  gc_DbmTranslation_fr_Text1195 : WSTRING(13) := "Dmc Heartbeat";
  gc_DbmTranslation_fr_Text1196 : WSTRING(15) := "Power On Ok Dmc";
  gc_DbmTranslation_fr_Text1197 : WSTRING(16) := "Operationnal Dmc";
  gc_DbmTranslation_fr_Text1198 : WSTRING(18) := "Go To Operationnal";
  gc_DbmTranslation_fr_Text1199 : WSTRING(22) := "New Go To Operationnal";
  gc_DbmTranslation_fr_Text1200 : WSTRING(16) := "Send Command NMT";
  gc_DbmTranslation_fr_Text1201 : WSTRING(12) := "Step Raz Dmc";
  gc_DbmTranslation_fr_Text1202 : WSTRING(24) := "Command Raz Dmc On Going";
  gc_DbmTranslation_fr_Text1203 : WSTRING(22) := "Dig4 Input Command STO";
  gc_DbmTranslation_fr_Text1204 : WSTRING(20) := "Active Fault Raz Dmc";
  gc_DbmTranslation_fr_Text1205 : WSTRING(16) := "Active Fault Dmc";
  gc_DbmTranslation_fr_Text1206 : WSTRING(30) := "Delta Arm Angular Sensor state";
  gc_DbmTranslation_fr_Text1207 : WSTRING(30) := "Delta Arm Angular Sensor value";
  gc_DbmTranslation_fr_Text1208 : WSTRING(56) := "Delta Arm Angular Sensor with calibration scaling  value";
  gc_DbmTranslation_fr_Text1209 : WSTRING(41) := "Delta Arm Angular Sensor raw value Master";
  gc_DbmTranslation_fr_Text1210 : WSTRING(40) := "Delta Arm Angular Sensor raw value slave";
  gc_DbmTranslation_fr_Text1211 : WSTRING(30) := "Arrow Arm Angular Sensor state";
  gc_DbmTranslation_fr_Text1212 : WSTRING(30) := "Arrow Arm Angular Sensor value";
  gc_DbmTranslation_fr_Text1213 : WSTRING(56) := "Arrow Arm Angular Sensor with calibration scaling  value";
  gc_DbmTranslation_fr_Text1214 : WSTRING(34) := "Arrow Arm Angular Sensor raw value";
  gc_DbmTranslation_fr_Text1215 : WSTRING(30) := "Arrow Arm Angular Sensor state";
  gc_DbmTranslation_fr_Text1216 : WSTRING(15) := "Gas Gauge value";
  gc_DbmTranslation_fr_Text1217 : WSTRING(19) := "Gas Gauge raw value";
  gc_DbmTranslation_fr_Text1218 : WSTRING(11) := "Aru 1 state";
  gc_DbmTranslation_fr_Text1219 : WSTRING(15) := "Aru 1 raw value";
  gc_DbmTranslation_fr_Text1220 : WSTRING(11) := "Aru 2 state";
  gc_DbmTranslation_fr_Text1221 : WSTRING(15) := "Aru 2 raw value";
  gc_DbmTranslation_fr_Text1222 : WSTRING(32) := "Entry Telescope Fdc Sensor state";
  gc_DbmTranslation_fr_Text1223 : WSTRING(36) := "Entry Telescope Fdc Sensor raw value";
  gc_DbmTranslation_fr_Text1224 : WSTRING(36) := "Folded Delta Arm Sensor state switch";
  gc_DbmTranslation_fr_Text1225 : WSTRING(33) := "Folded Delta Arm Sensor raw value";
  gc_DbmTranslation_fr_Text1226 : WSTRING(35) := "Folded Boom Arm Sensor state switch";
  gc_DbmTranslation_fr_Text1227 : WSTRING(32) := "Folded Boom Arm Sensor raw value";
  gc_DbmTranslation_fr_Text1228 : WSTRING(33) := "Forcing Motor Regime state switch";
  gc_DbmTranslation_fr_Text1229 : WSTRING(30) := "Forcing Motor Regime raw value";
  gc_DbmTranslation_fr_Text1230 : WSTRING(24) := "Active Help state switch";
  gc_DbmTranslation_fr_Text1231 : WSTRING(21) := "Active Help raw value";
  gc_DbmTranslation_fr_Text1232 : WSTRING(25) := "Oil Pressure state swtich";
  gc_DbmTranslation_fr_Text1233 : WSTRING(22) := "Oil Pressure raw value";
  gc_DbmTranslation_fr_Text1234 : WSTRING(30) := "Water Temperature state switch";
  gc_DbmTranslation_fr_Text1235 : WSTRING(27) := "Water Temperature raw value";
  gc_DbmTranslation_fr_Text1236 : WSTRING(21) := "Stop Motor Info State";
  gc_DbmTranslation_fr_Text1237 : WSTRING(25) := "Stop Motor Info Raw value";
  gc_DbmTranslation_fr_Text1238 : WSTRING(26) := "Turret Post Selector State";
  gc_DbmTranslation_fr_Text1239 : WSTRING(30) := "Turret Post Selector Raw Value";
  gc_DbmTranslation_fr_Text1240 : WSTRING(25) := "Radio Post Selector State";
  gc_DbmTranslation_fr_Text1241 : WSTRING(29) := "Radio Post Selector Raw Value";
  gc_DbmTranslation_fr_Text1242 : WSTRING(27) := "Nacelle Post Selector State";
  gc_DbmTranslation_fr_Text1243 : WSTRING(31) := "Nacelle Post Selector Raw Value";
  gc_DbmTranslation_fr_Text1244 : WSTRING(43) := "Regime motor alternator rotation per minute";
  gc_DbmTranslation_fr_Text1245 : WSTRING(26) := "Alternator charge ok state";
  gc_DbmTranslation_fr_Text1246 : WSTRING(26) := "Alternator charge ok value";
  gc_DbmTranslation_fr_Text1247 : WSTRING(35) := "Transmission1 Pressure Sensor State";
  gc_DbmTranslation_fr_Text1248 : WSTRING(35) := "Transmission1 Pressure Sensor Value";
  gc_DbmTranslation_fr_Text1249 : WSTRING(35) := "Transmission2 Pressure Sensor State";
  gc_DbmTranslation_fr_Text1250 : WSTRING(35) := "Transmission2 Pressure Sensor Value";
  gc_DbmTranslation_fr_Text1251 : WSTRING(25) := "Fault Pvg Delta Arm state";
  gc_DbmTranslation_fr_Text1252 : WSTRING(29) := "Fault Pvg Delta Arm raw value";
  gc_DbmTranslation_fr_Text1253 : WSTRING(24) := "Fault Pvg Boom Arm state";
  gc_DbmTranslation_fr_Text1254 : WSTRING(28) := "Fault Pvg Boom Arm raw value";
  gc_DbmTranslation_fr_Text1255 : WSTRING(29) := "Fault Pvg Telescope Arm state";
  gc_DbmTranslation_fr_Text1256 : WSTRING(33) := "Fault Pvg Telescope Arm raw value";
  gc_DbmTranslation_fr_Text1257 : WSTRING(26) := "Fault Pvg Ev Pro TOR state";
  gc_DbmTranslation_fr_Text1258 : WSTRING(30) := "Fault Pvg Ev Pro TOR raw value";
  gc_DbmTranslation_fr_Text1259 : WSTRING(28) := "Bypass Pressure Sensor State";
  gc_DbmTranslation_fr_Text1260 : WSTRING(28) := "Bypass Pressure Sensor Value";
  gc_DbmTranslation_fr_Text1261 : WSTRING(31) := "Bypass Pressure Sensor RawValue";
  gc_DbmTranslation_fr_Text1262 : WSTRING(19) := "Starter Motor State";
  gc_DbmTranslation_fr_Text1263 : WSTRING(23) := "Starter Motor Raw value";
  gc_DbmTranslation_fr_Text1264 : WSTRING(33) := "Oil Tank Temperature Sensor State";
  gc_DbmTranslation_fr_Text1265 : WSTRING(33) := "Oil Tank Temperature Sensor Value";
  gc_DbmTranslation_fr_Text1266 : WSTRING(37) := "Oil Tank Temperature Sensor Raw value";
  gc_DbmTranslation_fr_Text1267 : WSTRING(17) := "Blue Fire command";
  gc_DbmTranslation_fr_Text1268 : WSTRING(22) := "Blue Fire actual value";
  gc_DbmTranslation_fr_Text1269 : WSTRING(29) := "Orange Flashing Light command";
  gc_DbmTranslation_fr_Text1270 : WSTRING(34) := "Orange Flashing Light actual value";
  gc_DbmTranslation_fr_Text1271 : WSTRING(20) := "Anti Startup command";
  gc_DbmTranslation_fr_Text1272 : WSTRING(18) := "Anti Startup Value";
  gc_DbmTranslation_fr_Text1273 : WSTRING(18) := "Stop Motor command";
  gc_DbmTranslation_fr_Text1274 : WSTRING(15) := "Warming command";
  gc_DbmTranslation_fr_Text1275 : WSTRING(17) := "Ev Bypass command";
  gc_DbmTranslation_fr_Text1276 : WSTRING(21) := "EvBypass actual value";
  gc_DbmTranslation_fr_Text1277 : WSTRING(28) := "Supply Pvg Delta Arm command";
  gc_DbmTranslation_fr_Text1278 : WSTRING(33) := "Supply Pvg Delta Arm actual value";
  gc_DbmTranslation_fr_Text1279 : WSTRING(28) := "Supply Pvg Arrow Arm command";
  gc_DbmTranslation_fr_Text1280 : WSTRING(33) := "Supply Pvg Arrow Arm actual value";
  gc_DbmTranslation_fr_Text1281 : WSTRING(32) := "Supply Pvg Telescope Arm command";
  gc_DbmTranslation_fr_Text1282 : WSTRING(37) := "Supply Pvg Telescope Arm actual value";
  gc_DbmTranslation_fr_Text1283 : WSTRING(30) := "Supply Pvg Prop Ev TOR command";
  gc_DbmTranslation_fr_Text1284 : WSTRING(35) := "Supply Pvg Prop Ev TOR actual value";
  gc_DbmTranslation_fr_Text1285 : WSTRING(33) := "Ev Prop Motor Accelerator command";
  gc_DbmTranslation_fr_Text1286 : WSTRING(23) := "Ev Prop Generator state";
  gc_DbmTranslation_fr_Text1287 : WSTRING(25) := "Ev Prop Generator command";
  gc_DbmTranslation_fr_Text1288 : WSTRING(25) := "Ev Pro pGenerator current";
  gc_DbmTranslation_fr_Text1289 : WSTRING(16) := "Noisemaker state";
  gc_DbmTranslation_fr_Text1290 : WSTRING(18) := "Noisemaker command";
  gc_DbmTranslation_fr_Text1291 : WSTRING(41) := "Ev Rotation Turret Counter Clokwise state";
  gc_DbmTranslation_fr_Text1292 : WSTRING(48) := "Ev Rotation Turret Counter Clokwise command bool";
  gc_DbmTranslation_fr_Text1293 : WSTRING(33) := "Ev Rotation Turret Clokwise state";
  gc_DbmTranslation_fr_Text1294 : WSTRING(40) := "Ev Rotation Turret Clokwise command bool";
  gc_DbmTranslation_fr_Text1295 : WSTRING(41) := "Ev Rotation Basket Counter Clokwise state";
  gc_DbmTranslation_fr_Text1296 : WSTRING(51) := "Ev Rotation Basket counter clokwise command boolean";
  gc_DbmTranslation_fr_Text1297 : WSTRING(33) := "Ev Rotation Basket Clokwise state";
  gc_DbmTranslation_fr_Text1298 : WSTRING(43) := "Ev Rotation Basket clowkise command boolean";
  gc_DbmTranslation_fr_Text1299 : WSTRING(20) := "Ev Up Pendular state";
  gc_DbmTranslation_fr_Text1300 : WSTRING(27) := "Ev Up Pendular command bool";
  gc_DbmTranslation_fr_Text1301 : WSTRING(22) := "Ev Down Pendular state";
  gc_DbmTranslation_fr_Text1302 : WSTRING(29) := "Ev Down Pendular command bool";
  gc_DbmTranslation_fr_Text1303 : WSTRING(30) := "Ev Up Inclinaison Basket state";
  gc_DbmTranslation_fr_Text1304 : WSTRING(37) := "Ev Up Inclinaison Basket command bool";
  gc_DbmTranslation_fr_Text1305 : WSTRING(32) := "Ev Down Inclinaison Basket state";
  gc_DbmTranslation_fr_Text1306 : WSTRING(34) := "Ev Down Inclinaison Basket command";
  gc_DbmTranslation_fr_Text1307 : WSTRING(39) := "Ev Down Inclinaison Basket command bool";
  gc_DbmTranslation_fr_Text1308 : WSTRING(34) := "Ev Down Inclinaison Basket current";
  gc_DbmTranslation_fr_Text1309 : WSTRING(21) := "Pvg Delta Arm command";
  gc_DbmTranslation_fr_Text1310 : WSTRING(28) := "Pvg Delta Arm actual voltage";
  gc_DbmTranslation_fr_Text1311 : WSTRING(21) := "Pvg arrow Arm command";
  gc_DbmTranslation_fr_Text1312 : WSTRING(28) := "Pvg arrow Arm actual voltage";
  gc_DbmTranslation_fr_Text1313 : WSTRING(25) := "Pvg Arm Telescope command";
  gc_DbmTranslation_fr_Text1314 : WSTRING(32) := "Pvg Arm Telescope actual voltage";
  gc_DbmTranslation_fr_Text1315 : WSTRING(25) := "Overload Security Command";
  gc_DbmTranslation_fr_Text1316 : WSTRING(23) := "Overload Security Value";
  gc_DbmTranslation_fr_Text1317 : WSTRING(26) := "Suplly Tor Sensors Command";
  gc_DbmTranslation_fr_Text1318 : WSTRING(24) := "Suplly Tor Sensors Value";
  gc_DbmTranslation_fr_Text1319 : WSTRING(26) := "Suplly Ana Sensors Command";
  gc_DbmTranslation_fr_Text1320 : WSTRING(24) := "Suplly Ana Sensors Value";
  gc_DbmTranslation_fr_Text1321 : WSTRING(24) := "Ev Sync Rotation Command";
  gc_DbmTranslation_fr_Text1322 : WSTRING(22) := "Ev Sync Rotation Value";
  gc_DbmTranslation_fr_Text1323 : WSTRING(18) := "Pvg Ev Tor command";
  gc_DbmTranslation_fr_Text1324 : WSTRING(25) := "Pvg Ev Tor actual voltage";
  gc_DbmTranslation_fr_Text1325 : WSTRING(25) := "Ev Up pendular activation";
  gc_DbmTranslation_fr_Text1326 : WSTRING(27) := "Ev Down pendular activation";
  gc_DbmTranslation_fr_Text1327 : WSTRING(46) := "Ev rotation basket counter clokwise activation";
  gc_DbmTranslation_fr_Text1328 : WSTRING(38) := "Ev rotation basket clokwise activation";
  gc_DbmTranslation_fr_Text1329 : WSTRING(36) := "Ev Up inclinasison basket activation";
  gc_DbmTranslation_fr_Text1330 : WSTRING(38) := "Ev Down inclinasison basket activation";
  gc_DbmTranslation_fr_Text1331 : WSTRING(39) := "Ev rotation turret cloclwise activation";
  gc_DbmTranslation_fr_Text1332 : WSTRING(47) := "Ev rotation turret counter cloclwise activation";
  gc_DbmTranslation_fr_Text1333 : WSTRING(33) := "Ev Selector Rotation Turret State";
  gc_DbmTranslation_fr_Text1334 : WSTRING(35) := "Ev Selector Rotation Turret command";
  gc_DbmTranslation_fr_Text1335 : WSTRING(48) := "Return low side ev pro accelerator motor command";
  gc_DbmTranslation_fr_Text1336 : WSTRING(40) := "Return low side ev pro generator command";
  gc_DbmTranslation_fr_Text1337 : WSTRING(38) := "Return low side ev pro generator value";
  gc_DbmTranslation_fr_Text1338 : WSTRING(31) := "Ev Up Axle oscillant activation";
  gc_DbmTranslation_fr_Text1339 : WSTRING(33) := "Ev Down Axle oscillant activation";
  gc_DbmTranslation_fr_Text1340 : WSTRING(24) := "Ev Up Axle oscillant cmd";
  gc_DbmTranslation_fr_Text1341 : WSTRING(26) := "Ev Down Axle oscillant cmd";
  gc_DbmTranslation_fr_Text1342 : WSTRING(26) := "Ev Up Axle fixe activation";
  gc_DbmTranslation_fr_Text1343 : WSTRING(28) := "Ev Down Axle fixe activation";
  gc_DbmTranslation_fr_Text1344 : WSTRING(19) := "Ev Up Axle fixe cmd";
  gc_DbmTranslation_fr_Text1345 : WSTRING(21) := "Ev Down Axle fixe cmd";
  gc_DbmTranslation_fr_Text1346 : WSTRING(29) := "Ev Up Mast Measure Activation";
  gc_DbmTranslation_fr_Text1347 : WSTRING(22) := "Ev Up Mast Measure cmd";
  gc_DbmTranslation_fr_Text1348 : WSTRING(31) := "Ev down Mast Measure Activation";
  gc_DbmTranslation_fr_Text1349 : WSTRING(24) := "Ev down Mast Measure cmd";
  gc_DbmTranslation_fr_Text1350 : WSTRING(33) := "White light Av 15746 actual value";
  gc_DbmTranslation_fr_Text1351 : WSTRING(24) := "White light Av 15746 cmd";
  gc_DbmTranslation_fr_Text1352 : WSTRING(28) := "Ev crawler only actual value";
  gc_DbmTranslation_fr_Text1353 : WSTRING(19) := "Ev crawler only cmd";
  gc_DbmTranslation_fr_Text1354 : WSTRING(44) := "Relay electric Reload With Generator command";
  gc_DbmTranslation_fr_Text1355 : WSTRING(42) := "Relay electric Reload With Generator state";
  gc_DbmTranslation_fr_Text1356 : WSTRING(29) := "Ev Deviator movements command";
  gc_DbmTranslation_fr_Text1357 : WSTRING(27) := "Ev Deviator movements state";
  gc_DbmTranslation_fr_Text1358 : WSTRING(29) := "Ev Boost Regeneration command";
  gc_DbmTranslation_fr_Text1359 : WSTRING(27) := "Ev Boost Regeneration state";
  gc_DbmTranslation_fr_Text1360 : WSTRING(25) := "Byte increased each cycle";
  gc_DbmTranslation_fr_Text1361 : WSTRING(22) := "Watchdog current state";
  gc_DbmTranslation_fr_Text1362 : WSTRING(11) := "Ecu voltage";
  gc_DbmTranslation_fr_Text1363 : WSTRING(16) := "Bypass Arm Delta";
  gc_DbmTranslation_fr_Text1364 : WSTRING(16) := "Bypass Arm Arrow";
  gc_DbmTranslation_fr_Text1365 : WSTRING(20) := "Bypass Arm Telescope";
  gc_DbmTranslation_fr_Text1366 : WSTRING(23) := "test bool evision objet";
  gc_DbmTranslation_fr_Text1367 : WSTRING(42) := "Pvg consigne -10000 1000 to command output";
  gc_DbmTranslation_fr_Text1368 : WSTRING(58) := "Command Pvg Ev Tor for turret movement by joystick nacelle";
  gc_DbmTranslation_fr_Text1369 : WSTRING(19) := "Engine on run phase";
  gc_DbmTranslation_fr_Text1370 : WSTRING(0) := "";
  gc_DbmTranslation_fr_Text1371 : WSTRING(0) := "";
  gc_DbmTranslation_fr_Text1372 : WSTRING(0) := "";
  gc_DbmTranslation_fr_Text1373 : WSTRING(0) := "";
  gc_DbmTranslation_fr_Text1374 : WSTRING(0) := "";
  gc_DbmTranslation_fr_Text1375 : WSTRING(0) := "";
  gc_DbmTranslation_fr_Text1376 : WSTRING(50) := "Scaling value of joystick turret arm -10000 0 1000";
  gc_DbmTranslation_fr_Text1377 : WSTRING(49) := "Scaling value of joystick delta arm -10000 0 1000";
  gc_DbmTranslation_fr_Text1378 : WSTRING(54) := "Pvg Delta Arm Consigne apply to ramp to control output";
  gc_DbmTranslation_fr_Text1379 : WSTRING(49) := "Scaling value of joystick arrow arm -10000 0 1000";
  gc_DbmTranslation_fr_Text1380 : WSTRING(54) := "Pvg Arrow Arm Consigne apply to ramp to control output";
  gc_DbmTranslation_fr_Text1381 : WSTRING(53) := "Scaling value of joystick telescope arm -10000 0 1000";
  gc_DbmTranslation_fr_Text1382 : WSTRING(58) := "Pvg telescope Arm Consigne apply to ramp to control output";
  gc_DbmTranslation_fr_Text1383 : WSTRING(30) := "Range value of pvg tor min max";
  gc_DbmTranslation_fr_Text1384 : WSTRING(30) := "Range value of pvg tor min max";
  gc_DbmTranslation_fr_Text1385 : WSTRING(30) := "Range value of pvg tor min max";
  gc_DbmTranslation_fr_Text1386 : WSTRING(30) := "Range value of pvg tor min max";
  gc_DbmTranslation_fr_Text1387 : WSTRING(30) := "Range value of pvg tor min max";
  gc_DbmTranslation_fr_Text1388 : WSTRING(30) := "Range value of pvg tor min max";
  gc_DbmTranslation_fr_Text1389 : WSTRING(25) := "Active bool just for test";
  gc_DbmTranslation_fr_Text1390 : WSTRING(32) := "Portilon close and ladder folded";
  gc_DbmTranslation_fr_Text1391 : WSTRING(14) := "Active Failure";
  gc_DbmTranslation_fr_Text1392 : WSTRING(43) := "Condition to stop all movement nacelle post";
  gc_DbmTranslation_fr_Text1393 : WSTRING(18) := "Average Time cycle";
  gc_DbmTranslation_fr_Text1394 : WSTRING(14) := "Max time cycle";
  gc_DbmTranslation_fr_Text1395 : WSTRING(0) := "";
  gc_DbmTranslation_fr_Text1396 : WSTRING(16) := "Lynx On All Mvts";
  gc_DbmTranslation_fr_Text1397 : WSTRING(31) := "Return value of start 48xs func";
  gc_DbmTranslation_fr_Text1398 : WSTRING(34) := "Index version of 48XS slave module";
  gc_DbmTranslation_fr_Text1399 : WSTRING(38) := "Shunt all logic to test electricall IO";
  gc_DbmTranslation_fr_Text1400 : WSTRING(21) := "Major version of 48xs";
  gc_DbmTranslation_fr_Text1401 : WSTRING(21) := "Minor version of 48xs";
  gc_DbmTranslation_fr_Text1402 : WSTRING(20) := "Path version of 48xs";
  gc_DbmTranslation_fr_Text1403 : WSTRING(22) := "Custom version of 48xs";
  gc_DbmTranslation_fr_Text1404 : WSTRING(19) := "Running Stable 48XS";
  gc_DbmTranslation_fr_Text1405 : WSTRING(12) := "Low Blinking";
  gc_DbmTranslation_fr_Text1406 : WSTRING(17) := "Diag Faulty Value";
  gc_DbmTranslation_fr_Text1407 : WSTRING(15) := "Diag Device Num";
  gc_DbmTranslation_fr_Text1408 : WSTRING(15) := "Diag Error Code";
  gc_DbmTranslation_fr_Text1409 : WSTRING(21) := "Engine running stable";
  gc_DbmTranslation_fr_Text1410 : WSTRING(19) := "Bypass test command";
  gc_DbmTranslation_fr_Text1411 : WSTRING(37) := "Portillon is installed on the machine";
  gc_DbmTranslation_fr_Text1412 : WSTRING(34) := "Ladder is installed on the machine";
  gc_DbmTranslation_fr_Text1413 : WSTRING(41) := "Measuring mat is installed on the machine";
  gc_DbmTranslation_fr_Text1414 : WSTRING(64) := "The digital display o the measuring mast is used on this vehicle";
  gc_DbmTranslation_fr_Text1415 : WSTRING(35) := "Genetor is installed on the machine";
  gc_DbmTranslation_fr_Text1416 : WSTRING(29) := "Flashing light on rail option";
  gc_DbmTranslation_fr_Text1417 : WSTRING(55) := "Allow turret rotation beyond 135deg with automatic stop";
  gc_DbmTranslation_fr_Text1418 : WSTRING(20) := "Lynx On All Movement";
  gc_DbmTranslation_fr_Text1419 : WSTRING(46) := "White lights 15746 is installed on the machine";
  gc_DbmTranslation_fr_Text1420 : WSTRING(29) := "Autorisation Work key present";
  gc_DbmTranslation_fr_Text1421 : WSTRING(43) := "Option feu à éclat permanent pour Australie";
  gc_DbmTranslation_fr_Text1422 : WSTRING(56) := "Option for utilisation of the mast for electrified track";
  gc_DbmTranslation_fr_Text1423 : WSTRING(24) := "Presence of contact mast";
  gc_DbmTranslation_fr_Text1424 : WSTRING(0) := "";
  gc_DbmTranslation_fr_Text1425 : WSTRING(0) := "";
  gc_DbmTranslation_fr_Text1426 : WSTRING(0) := "";
  gc_DbmTranslation_fr_Text1427 : WSTRING(0) := "";
  gc_DbmTranslation_fr_Text1428 : WSTRING(0) := "";
  gc_DbmTranslation_fr_Text1429 : WSTRING(0) := "";
  gc_DbmTranslation_fr_Text1430 : WSTRING(0) := "";
  gc_DbmTranslation_fr_Text1431 : WSTRING(0) := "";
  gc_DbmTranslation_fr_Text1432 : WSTRING(0) := "";
  gc_DbmTranslation_fr_Text1433 : WSTRING(0) := "";
  gc_DbmTranslation_fr_Text1434 : WSTRING(0) := "";
  gc_DbmTranslation_fr_Text1435 : WSTRING(0) := "";
  gc_DbmTranslation_fr_Text1436 : WSTRING(0) := "";
  gc_DbmTranslation_fr_Text1437 : WSTRING(0) := "";
  gc_DbmTranslation_fr_Text1438 : WSTRING(0) := "";
  gc_DbmTranslation_fr_Text1439 : WSTRING(42) := "Reject counter of reloading with generator";
  gc_DbmTranslation_fr_Text1440 : WSTRING(34) := "First Key no reload with generator";
  gc_DbmTranslation_fr_Text1441 : WSTRING(34) := "New Soc Uper Reload With Generator";
  gc_DbmTranslation_fr_Text1442 : WSTRING(33) := "Total regeneration time in minute";
  gc_DbmTranslation_fr_Text1443 : WSTRING(28) := "Total electric motor minutes";
  gc_DbmTranslation_fr_Text1444 : WSTRING(75) := "Pvg Up Delta Arm turret post command in pourcent regarding batterie voltage";
  gc_DbmTranslation_fr_Text1445 : WSTRING(77) := "Pvg Down Delta Arm turret post command in pourcent regarding batterie voltage";
  gc_DbmTranslation_fr_Text1446 : WSTRING(75) := "Pvg Up Arrow Arm turret post command in pourcent regarding batterie voltage";
  gc_DbmTranslation_fr_Text1447 : WSTRING(77) := "Pvg Down Arrow Arm turret post command in pourcent regarding batterie voltage";
  gc_DbmTranslation_fr_Text1448 : WSTRING(79) := "Pvg In Telescope Arm turret post command in pourcent regarding batterie voltage";
  gc_DbmTranslation_fr_Text1449 : WSTRING(80) := "Pvg Out Telescope Arm turret post command in pourcent regarding batterie voltage";
  gc_DbmTranslation_fr_Text1450 : WSTRING(89) := "Consigne max Pvg Up Delta Arm Nacelle post command in pourcent regarding batterie voltage";
  gc_DbmTranslation_fr_Text1451 : WSTRING(91) := "Consigne max Pvg Down Delta Arm Nacelle post command in pourcent regarding batterie voltage";
  gc_DbmTranslation_fr_Text1452 : WSTRING(89) := "Consigne max Pvg Up Arrow Arm Nacelle post command in pourcent regarding batterie voltage";
  gc_DbmTranslation_fr_Text1453 : WSTRING(91) := "Consigne max Pvg Down Arrow Arm Nacelle post command in pourcent regarding batterie voltage";
  gc_DbmTranslation_fr_Text1454 : WSTRING(93) := "Consigne max Pvg in Telescope Arm Nacelle post command in pourcent regarding batterie voltage";
  gc_DbmTranslation_fr_Text1455 : WSTRING(94) := "Consigne max Pvg out Telescope Arm Nacelle post command in pourcent regarding batterie voltage";
  gc_DbmTranslation_fr_Text1456 : WSTRING(97) := "Consigne min Pvg to move Up Delta Arm Nacelle post command in pourcent regarding batterie voltage";
  gc_DbmTranslation_fr_Text1457 : WSTRING(99) := "Consigne min Pvg to move Down Delta Arm Nacelle post command in pourcent regarding batterie voltage";
  gc_DbmTranslation_fr_Text1458 : WSTRING(97) := "Consigne min Pvg to move Up Arrow Arm Nacelle post command in pourcent regarding batterie voltage";
  gc_DbmTranslation_fr_Text1459 : WSTRING(99) := "Consigne min Pvg to move Down Arrow Arm Nacelle post command in pourcent regarding batterie voltage";
  gc_DbmTranslation_fr_Text1460 : WSTRING(101) := "Consigne min Pvg to move In Telescope Arm Nacelle post command in pourcent regarding batterie voltage";
  gc_DbmTranslation_fr_Text1461 : WSTRING(102) := "Consigne min Pvg to move Out Telescope Arm Nacelle post command in pourcent regarding batterie voltage";
  gc_DbmTranslation_fr_Text1462 : WSTRING(36) := "Treshold Ana to bool input from 48xs";
  gc_DbmTranslation_fr_Text1463 : WSTRING(61) := "Pvg axle movement command pourcent regarding batterie voltage";
  gc_DbmTranslation_fr_Text1464 : WSTRING(25) := "Dead zone joystick turret";
  gc_DbmTranslation_fr_Text1465 : WSTRING(28) := "Dead zone joystick delta arm";
  gc_DbmTranslation_fr_Text1466 : WSTRING(27) := "Dead zone joystick telescop";
  gc_DbmTranslation_fr_Text1467 : WSTRING(24) := "Dead Zone joystick arrow";
  gc_DbmTranslation_fr_Text1468 : WSTRING(35) := "Dead Zone joystick rail advancement";
  gc_DbmTranslation_fr_Text1469 : WSTRING(34) := "Dead Zone joystick rotation turret";
  gc_DbmTranslation_fr_Text1470 : WSTRING(66) := "EvPropMotorAccelerator - PWM output parameters- engine off current";
  gc_DbmTranslation_fr_Text1471 : WSTRING(63) := "EvPropMotorAccelerator - PWM output parameters- minimal current";
  gc_DbmTranslation_fr_Text1472 : WSTRING(61) := "EvPropMotorAccelerator - PWM output parameters- stop current ";
  gc_DbmTranslation_fr_Text1473 : WSTRING(59) := "EvPropGenerator - PWM output parameters- engine off current";
  gc_DbmTranslation_fr_Text1474 : WSTRING(55) := "EvPropGenerator- PWM output parameters- minimal current";
  gc_DbmTranslation_fr_Text1475 : WSTRING(53) := "EvPropGenerator- PWM output parameters- stop current ";
  gc_DbmTranslation_fr_Text1476 : WSTRING(56) := "PID - Ev Prop Motor Accelerator - Gp - proportional gain";
  gc_DbmTranslation_fr_Text1477 : WSTRING(64) := "PID - Ev Prop Motor Accelerator - Ti - integration time constant";
  gc_DbmTranslation_fr_Text1478 : WSTRING(63) := "PID - Ev Prop Motor Accelerator - Td - derivation time constant";
  gc_DbmTranslation_fr_Text1479 : WSTRING(48) := "PID - Ev Prop Generator - Gp - proportional gain";
  gc_DbmTranslation_fr_Text1480 : WSTRING(55) := "PID - Ev Prop Generator- Ti - integration time constant";
  gc_DbmTranslation_fr_Text1481 : WSTRING(55) := "PID - Ev Prop Generator - Td - derivation time constant";
  gc_DbmTranslation_fr_Text1482 : WSTRING(67) := "Deviation Limit beetween 2 signals for transmission pressure sensor";
  gc_DbmTranslation_fr_Text1483 : WSTRING(71) := "DeltaArmAngularSensor - input current - output characteristic - Positif";
  gc_DbmTranslation_fr_Text1484 : WSTRING(71) := "DeltaArmAngularSensor - input current - output characteristic - Neutral";
  gc_DbmTranslation_fr_Text1485 : WSTRING(71) := "DeltaArmAngularSensor - input current - output characteristic - Negatif";
  gc_DbmTranslation_fr_Text1486 : WSTRING(61) := "Deviation Limit beetween 2 signals for delta arm angle sensor";
  gc_DbmTranslation_fr_Text1487 : WSTRING(71) := "ArrowArmAngularSensor - input current - output characteristic - Positif";
  gc_DbmTranslation_fr_Text1488 : WSTRING(71) := "ArrowArmAngularSensor - input current - output characteristic - Neutral";
  gc_DbmTranslation_fr_Text1489 : WSTRING(71) := "ArrowArmAngularSensor - input current - output characteristic - Negatif";
  gc_DbmTranslation_fr_Text1490 : WSTRING(61) := "Deviation Limit beetween 2 signals for arrow arm angle sensor";
  gc_DbmTranslation_fr_Text1491 : WSTRING(75) := "Min pvg up pendular with turret post in pourcent regarding batterie voltage";
  gc_DbmTranslation_fr_Text1492 : WSTRING(76) := "Min pvg up pendular with Nacelle post in pourcent regarding batterie voltage";
  gc_DbmTranslation_fr_Text1493 : WSTRING(74) := "Min pvg up pendular with Radio post in pourcent regarding batterie voltage";
  gc_DbmTranslation_fr_Text1494 : WSTRING(75) := "Max pvg up pendular with turret post in pourcent regarding batterie voltage";
  gc_DbmTranslation_fr_Text1495 : WSTRING(76) := "Max pvg up pendular with Nacelle post in pourcent regarding batterie voltage";
  gc_DbmTranslation_fr_Text1496 : WSTRING(74) := "Max pvg up pendular with Radio post in pourcent regarding batterie voltage";
  gc_DbmTranslation_fr_Text1497 : WSTRING(105) := "Ratio apply to ramp signal to control Pvg Ev Tor when up pendular movement is sollicited with turret post";
  gc_DbmTranslation_fr_Text1498 : WSTRING(105) := "Ratio apply to ramp signal to control Pvg Ev Tor when up pendular movement is sollicited with turret post";
  gc_DbmTranslation_fr_Text1499 : WSTRING(105) := "Ratio apply to ramp signal to control Pvg Ev Tor when up pendular movement is sollicited with turret post";
  gc_DbmTranslation_fr_Text1500 : WSTRING(106) := "Ratio apply to ramp signal to control Pvg Ev Tor when up pendular movement is sollicited with nacelle post";
  gc_DbmTranslation_fr_Text1501 : WSTRING(106) := "Ratio apply to ramp signal to control Pvg Ev Tor when up pendular movement is sollicited with nacelle post";
  gc_DbmTranslation_fr_Text1502 : WSTRING(106) := "Ratio apply to ramp signal to control Pvg Ev Tor when up pendular movement is sollicited with nacelle post";
  gc_DbmTranslation_fr_Text1503 : WSTRING(104) := "Ratio apply to ramp signal to control Pvg Ev Tor when up pendular movement is sollicited with radio post";
  gc_DbmTranslation_fr_Text1504 : WSTRING(104) := "Ratio apply to ramp signal to control Pvg Ev Tor when up pendular movement is sollicited with radio post";
  gc_DbmTranslation_fr_Text1505 : WSTRING(104) := "Ratio apply to ramp signal to control Pvg Ev Tor when up pendular movement is sollicited with radio post";
  gc_DbmTranslation_fr_Text1506 : WSTRING(77) := "Min pvg down pendular with turret post in pourcent regarding batterie voltage";
  gc_DbmTranslation_fr_Text1507 : WSTRING(78) := "Min pvg down pendular with Nacelle post in pourcent regarding batterie voltage";
  gc_DbmTranslation_fr_Text1508 : WSTRING(76) := "Min pvg down pendular with Radio post in pourcent regarding batterie voltage";
  gc_DbmTranslation_fr_Text1509 : WSTRING(77) := "Max pvg down pendular with turret post in pourcent regarding batterie voltage";
  gc_DbmTranslation_fr_Text1510 : WSTRING(78) := "Max pvg down pendular with Nacelle post in pourcent regarding batterie voltage";
  gc_DbmTranslation_fr_Text1511 : WSTRING(76) := "Max pvg down pendular with Radio post in pourcent regarding batterie voltage";
  gc_DbmTranslation_fr_Text1512 : WSTRING(107) := "Ratio apply to ramp signal to control Pvg Ev Tor when down pendular movement is sollicited with turret post";
  gc_DbmTranslation_fr_Text1513 : WSTRING(107) := "Ratio apply to ramp signal to control Pvg Ev Tor when down pendular movement is sollicited with turret post";
  gc_DbmTranslation_fr_Text1514 : WSTRING(107) := "Ratio apply to ramp signal to control Pvg Ev Tor when down pendular movement is sollicited with turret post";
  gc_DbmTranslation_fr_Text1515 : WSTRING(108) := "Ratio apply to ramp signal to control Pvg Ev Tor when down pendular movement is sollicited with nacelle post";
  gc_DbmTranslation_fr_Text1516 : WSTRING(108) := "Ratio apply to ramp signal to control Pvg Ev Tor when down pendular movement is sollicited with nacelle post";
  gc_DbmTranslation_fr_Text1517 : WSTRING(108) := "Ratio apply to ramp signal to control Pvg Ev Tor when down pendular movement is sollicited with nacelle post";
  gc_DbmTranslation_fr_Text1518 : WSTRING(106) := "Ratio apply to ramp signal to control Pvg Ev Tor when down pendular movement is sollicited with radio post";
  gc_DbmTranslation_fr_Text1519 : WSTRING(106) := "Ratio apply to ramp signal to control Pvg Ev Tor when down pendular movement is sollicited with radio post";
  gc_DbmTranslation_fr_Text1520 : WSTRING(106) := "Ratio apply to ramp signal to control Pvg Ev Tor when down pendular movement is sollicited with radio post";
  gc_DbmTranslation_fr_Text1521 : WSTRING(85) := "Min pvg up inclinaison basket with turret post in pourcent regarding batterie voltage";
  gc_DbmTranslation_fr_Text1522 : WSTRING(86) := "Min pvg up inclinaison basket with Nacelle post in pourcent regarding batterie voltage";
  gc_DbmTranslation_fr_Text1523 : WSTRING(84) := "Min pvg up inclinaison basket with Radio post in pourcent regarding batterie voltage";
  gc_DbmTranslation_fr_Text1524 : WSTRING(85) := "Max pvg up inclinaison basket with turret post in pourcent regarding batterie voltage";
  gc_DbmTranslation_fr_Text1525 : WSTRING(86) := "Max pvg up inclinaison basket with Nacelle post in pourcent regarding batterie voltage";
  gc_DbmTranslation_fr_Text1526 : WSTRING(84) := "Max pvg up inclinaison basket with Radio post in pourcent regarding batterie voltage";
  gc_DbmTranslation_fr_Text1527 : WSTRING(107) := "Ratio apply to ramp signal to Pvg Ev Tor when up inclinaison basket movement is sollicited with turret post";
  gc_DbmTranslation_fr_Text1528 : WSTRING(107) := "Ratio apply to ramp signal to Pvg Ev Tor when up inclinaison basket movement is sollicited with turret post";
  gc_DbmTranslation_fr_Text1529 : WSTRING(107) := "Ratio apply to ramp signal to Pvg Ev Tor when up inclinaison basket movement is sollicited with turret post";
  gc_DbmTranslation_fr_Text1530 : WSTRING(108) := "Ratio apply to ramp signal to Pvg Ev Tor when up inclinaison basket movement is sollicited with nacelle post";
  gc_DbmTranslation_fr_Text1531 : WSTRING(108) := "Ratio apply to ramp signal to Pvg Ev Tor when up inclinaison basket movement is sollicited with nacelle post";
  gc_DbmTranslation_fr_Text1532 : WSTRING(108) := "Ratio apply to ramp signal to Pvg Ev Tor when up inclinaison basket movement is sollicited with nacelle post";
  gc_DbmTranslation_fr_Text1533 : WSTRING(106) := "Ratio apply to ramp signal to Pvg Ev Tor when up inclinaison basket movement is sollicited with radio post";
  gc_DbmTranslation_fr_Text1534 : WSTRING(106) := "Ratio apply to ramp signal to Pvg Ev Tor when up inclinaison basket movement is sollicited with radio post";
  gc_DbmTranslation_fr_Text1535 : WSTRING(106) := "Ratio apply to ramp signal to Pvg Ev Tor when up inclinaison basket movement is sollicited with radio post";
  gc_DbmTranslation_fr_Text1536 : WSTRING(87) := "Min pvg down inclinaison basket with turret post in pourcent regarding batterie voltage";
  gc_DbmTranslation_fr_Text1537 : WSTRING(88) := "Min pvg down inclinaison basket with Nacelle post in pourcent regarding batterie voltage";
  gc_DbmTranslation_fr_Text1538 : WSTRING(86) := "Min pvg down inclinaison basket with Radio post in pourcent regarding batterie voltage";
  gc_DbmTranslation_fr_Text1539 : WSTRING(87) := "Max pvg down inclinaison basket with turret post in pourcent regarding batterie voltage";
  gc_DbmTranslation_fr_Text1540 : WSTRING(88) := "Max pvg down inclinaison basket with Nacelle post in pourcent regarding batterie voltage";
  gc_DbmTranslation_fr_Text1541 : WSTRING(86) := "Max pvg down inclinaison basket with Radio post in pourcent regarding batterie voltage";
  gc_DbmTranslation_fr_Text1542 : WSTRING(105) := "Ratio apply to ramp signal to Pvg Ev Tor when down inclinaison basket movement is sollicited with turret ";
  gc_DbmTranslation_fr_Text1543 : WSTRING(105) := "Ratio apply to ramp signal to Pvg Ev Tor when down inclinaison basket movement is sollicited with turret ";
  gc_DbmTranslation_fr_Text1544 : WSTRING(105) := "Ratio apply to ramp signal to Pvg Ev Tor when down inclinaison basket movement is sollicited with turret ";
  gc_DbmTranslation_fr_Text1545 : WSTRING(106) := "Ratio apply to ramp signal to Pvg Ev Tor when down inclinaison basket movement is sollicited with nacelle ";
  gc_DbmTranslation_fr_Text1546 : WSTRING(106) := "Ratio apply to ramp signal to Pvg Ev Tor when down inclinaison basket movement is sollicited with nacelle ";
  gc_DbmTranslation_fr_Text1547 : WSTRING(106) := "Ratio apply to ramp signal to Pvg Ev Tor when down inclinaison basket movement is sollicited with nacelle ";
  gc_DbmTranslation_fr_Text1548 : WSTRING(104) := "Ratio apply to ramp signal to Pvg Ev Tor when down inclinaison basket movement is sollicited with radio ";
  gc_DbmTranslation_fr_Text1549 : WSTRING(104) := "Ratio apply to ramp signal to Pvg Ev Tor when down inclinaison basket movement is sollicited with radio ";
  gc_DbmTranslation_fr_Text1550 : WSTRING(104) := "Ratio apply to ramp signal to Pvg Ev Tor when down inclinaison basket movement is sollicited with radio ";
  gc_DbmTranslation_fr_Text1551 : WSTRING(89) := "Min pvg rotation clockwise basket with turret post in pourcent regarding batterie voltage";
  gc_DbmTranslation_fr_Text1552 : WSTRING(90) := "Min pvg rotation clockwise basket with Nacelle post in pourcent regarding batterie voltage";
  gc_DbmTranslation_fr_Text1553 : WSTRING(88) := "Min pvg rotation clockwise basket with Radio post in pourcent regarding batterie voltage";
  gc_DbmTranslation_fr_Text1554 : WSTRING(89) := "Max pvg rotation clockwise basket with turret post in pourcent regarding batterie voltage";
  gc_DbmTranslation_fr_Text1555 : WSTRING(90) := "Max pvg rotation clockwise basket with Nacelle post in pourcent regarding batterie voltage";
  gc_DbmTranslation_fr_Text1556 : WSTRING(88) := "Max pvg rotation clockwise basket with Radio post in pourcent regarding batterie voltage";
  gc_DbmTranslation_fr_Text1557 : WSTRING(108) := "Ratio apply to ramp signal to control Pvg Ev Tor rotation clk basket movement is sollicited with radio nacel";
  gc_DbmTranslation_fr_Text1558 : WSTRING(108) := "Ratio apply to ramp signal to control Pvg Ev Tor rotation clk basket movement is sollicited with radio nacel";
  gc_DbmTranslation_fr_Text1559 : WSTRING(108) := "Ratio apply to ramp signal to control Pvg Ev Tor rotation clk basket movement is sollicited with radio nacel";
  gc_DbmTranslation_fr_Text1560 : WSTRING(108) := "Ratio apply to ramp signal to control Pvg Ev Tor rotation clk basket movement is sollicited with radio nacel";
  gc_DbmTranslation_fr_Text1561 : WSTRING(108) := "Ratio apply to ramp signal to control Pvg Ev Tor rotation clk basket movement is sollicited with radio nacel";
  gc_DbmTranslation_fr_Text1562 : WSTRING(108) := "Ratio apply to ramp signal to control Pvg Ev Tor rotation clk basket movement is sollicited with radio nacel";
  gc_DbmTranslation_fr_Text1563 : WSTRING(109) := "Ratio apply to ramp signal to control Pvg Ev Tor rotation clk basket movement is sollicited  with radio radio";
  gc_DbmTranslation_fr_Text1564 : WSTRING(109) := "Ratio apply to ramp signal to control Pvg Ev Tor rotation clk basket movement is sollicited  with radio radio";
  gc_DbmTranslation_fr_Text1565 : WSTRING(109) := "Ratio apply to ramp signal to control Pvg Ev Tor rotation clk basket movement is sollicited  with radio radio";
  gc_DbmTranslation_fr_Text1566 : WSTRING(97) := "Min pvg rotation counter clockwise basket with turret post in pourcent regarding batterie voltage";
  gc_DbmTranslation_fr_Text1567 : WSTRING(98) := "Min pvg rotation counter clockwise basket with Nacelle post in pourcent regarding batterie voltage";
  gc_DbmTranslation_fr_Text1568 : WSTRING(96) := "Min pvg rotation counter clockwise basket with Radio post in pourcent regarding batterie voltage";
  gc_DbmTranslation_fr_Text1569 : WSTRING(97) := "Max pvg rotation counter clockwise basket with turret post in pourcent regarding batterie voltage";
  gc_DbmTranslation_fr_Text1570 : WSTRING(98) := "Max pvg rotation counter clockwise basket with Nacelle post in pourcent regarding batterie voltage";
  gc_DbmTranslation_fr_Text1571 : WSTRING(96) := "Max pvg rotation counter clockwise basket with Radio post in pourcent regarding batterie voltage";
  gc_DbmTranslation_fr_Text1572 : WSTRING(109) := "Ratio apply to ramp signal to control Pvg Ev Tor rotation counter clockwise basket is sollicited with turret ";
  gc_DbmTranslation_fr_Text1573 : WSTRING(109) := "Ratio apply to ramp signal to control Pvg Ev Tor rotation counter clockwise basket is sollicited with turret ";
  gc_DbmTranslation_fr_Text1574 : WSTRING(109) := "Ratio apply to ramp signal to control Pvg Ev Tor rotation counter clockwise basket is sollicited with turret ";
  gc_DbmTranslation_fr_Text1575 : WSTRING(108) := "Ratio apply to ramp signal to control Pvg Ev Tor rotation counter clockwise basket is sollicited with nacel ";
  gc_DbmTranslation_fr_Text1576 : WSTRING(108) := "Ratio apply to ramp signal to control Pvg Ev Tor rotation counter clockwise basket is sollicited with nacel ";
  gc_DbmTranslation_fr_Text1577 : WSTRING(108) := "Ratio apply to ramp signal to control Pvg Ev Tor rotation counter clockwise basket is sollicited with nacel ";
  gc_DbmTranslation_fr_Text1578 : WSTRING(103) := "Ratio apply to ramp signal to Pvg Ev Tor rotation counter clk basket movement is sollicited with radio ";
  gc_DbmTranslation_fr_Text1579 : WSTRING(103) := "Ratio apply to ramp signal to Pvg Ev Tor rotation counter clk basket movement is sollicited with radio ";
  gc_DbmTranslation_fr_Text1580 : WSTRING(103) := "Ratio apply to ramp signal to Pvg Ev Tor rotation counter clk basket movement is sollicited with radio ";
  gc_DbmTranslation_fr_Text1581 : WSTRING(89) := "Min pvg rotation clockwise basket with turret post in pourcent regarding batterie voltage";
  gc_DbmTranslation_fr_Text1582 : WSTRING(90) := "Min pvg rotation clockwise basket with Nacelle post in pourcent regarding batterie voltage";
  gc_DbmTranslation_fr_Text1583 : WSTRING(88) := "Min pvg rotation clockwise basket with Radio post in pourcent regarding batterie voltage";
  gc_DbmTranslation_fr_Text1584 : WSTRING(89) := "Max pvg rotation clockwise basket with turret post in pourcent regarding batterie voltage";
  gc_DbmTranslation_fr_Text1585 : WSTRING(90) := "Max pvg rotation clockwise basket with Nacelle post in pourcent regarding batterie voltage";
  gc_DbmTranslation_fr_Text1586 : WSTRING(88) := "Max pvg rotation clockwise basket with Radio post in pourcent regarding batterie voltage";
  gc_DbmTranslation_fr_Text1587 : WSTRING(106) := "Ratio apply to ramp signal to Pvg Ev Tor rotation clockwise basket movement is sollicited with turret post";
  gc_DbmTranslation_fr_Text1588 : WSTRING(106) := "Ratio apply to ramp signal to Pvg Ev Tor rotation clockwise basket movement is sollicited with turret post";
  gc_DbmTranslation_fr_Text1589 : WSTRING(106) := "Ratio apply to ramp signal to Pvg Ev Tor rotation clockwise basket movement is sollicited with turret post";
  gc_DbmTranslation_fr_Text1590 : WSTRING(107) := "Ratio apply to ramp signal to Pvg Ev Tor rotation clockwise basket movement is sollicited with Nacelle post";
  gc_DbmTranslation_fr_Text1591 : WSTRING(107) := "Ratio apply to ramp signal to Pvg Ev Tor rotation clockwise basket movement is sollicited with Nacelle post";
  gc_DbmTranslation_fr_Text1592 : WSTRING(107) := "Ratio apply to ramp signal to Pvg Ev Tor rotation clockwise basket movement is sollicited with Nacelle post";
  gc_DbmTranslation_fr_Text1593 : WSTRING(105) := "Ratio apply to ramp signal to Pvg Ev Tor rotation clockwise basket movement is sollicited with radio post";
  gc_DbmTranslation_fr_Text1594 : WSTRING(105) := "Ratio apply to ramp signal to Pvg Ev Tor rotation clockwise basket movement is sollicited with radio post";
  gc_DbmTranslation_fr_Text1595 : WSTRING(105) := "Ratio apply to ramp signal to Pvg Ev Tor rotation clockwise basket movement is sollicited with radio post";
  gc_DbmTranslation_fr_Text1596 : WSTRING(97) := "Min pvg rotation counter clockwise basket with turret post in pourcent regarding batterie voltage";
  gc_DbmTranslation_fr_Text1597 : WSTRING(98) := "Min pvg rotation counter clockwise basket with Nacelle post in pourcent regarding batterie voltage";
  gc_DbmTranslation_fr_Text1598 : WSTRING(96) := "Min pvg rotation counter clockwise basket with Radio post in pourcent regarding batterie voltage";
  gc_DbmTranslation_fr_Text1599 : WSTRING(97) := "Max pvg rotation counter clockwise basket with turret post in pourcent regarding batterie voltage";
  gc_DbmTranslation_fr_Text1600 : WSTRING(98) := "Max pvg rotation counter clockwise basket with Nacelle post in pourcent regarding batterie voltage";
  gc_DbmTranslation_fr_Text1601 : WSTRING(96) := "Max pvg rotation counter clockwise basket with Radio post in pourcent regarding batterie voltage";
  gc_DbmTranslation_fr_Text1602 : WSTRING(110) := "Ratio apply to ramp signal to Pvg Ev Tor rotation counter clockwise basket movement is sollicited with turret ";
  gc_DbmTranslation_fr_Text1603 : WSTRING(110) := "Ratio apply to ramp signal to Pvg Ev Tor rotation counter clockwise basket movement is sollicited with turret ";
  gc_DbmTranslation_fr_Text1604 : WSTRING(110) := "Ratio apply to ramp signal to Pvg Ev Tor rotation counter clockwise basket movement is sollicited with turret ";
  gc_DbmTranslation_fr_Text1605 : WSTRING(111) := "Ratio apply to ramp signal to Pvg Ev Tor rotation counter clockwise basket movement is sollicited with nacelle ";
  gc_DbmTranslation_fr_Text1606 : WSTRING(111) := "Ratio apply to ramp signal to Pvg Ev Tor rotation counter clockwise basket movement is sollicited with nacelle ";
  gc_DbmTranslation_fr_Text1607 : WSTRING(111) := "Ratio apply to ramp signal to Pvg Ev Tor rotation counter clockwise basket movement is sollicited with nacelle ";
  gc_DbmTranslation_fr_Text1608 : WSTRING(109) := "Ratio apply to ramp signal to Pvg Ev Tor rotation counter clockwise basket movement is sollicited with radio ";
  gc_DbmTranslation_fr_Text1609 : WSTRING(109) := "Ratio apply to ramp signal to Pvg Ev Tor rotation counter clockwise basket movement is sollicited with radio ";
  gc_DbmTranslation_fr_Text1610 : WSTRING(109) := "Ratio apply to ramp signal to Pvg Ev Tor rotation counter clockwise basket movement is sollicited with radio ";
  gc_DbmTranslation_fr_Text1611 : WSTRING(25) := "Min pvg up axle oscillant";
  gc_DbmTranslation_fr_Text1612 : WSTRING(25) := "Max pvg up axle oscillant";
  gc_DbmTranslation_fr_Text1613 : WSTRING(94) := "Ratio apply to ramp signal to control Pvg Ev Tor when up axle oscillant movement is sollicited";
  gc_DbmTranslation_fr_Text1614 : WSTRING(94) := "Ratio apply to ramp signal to control Pvg Ev Tor when up axle oscillant movement is sollicited";
  gc_DbmTranslation_fr_Text1615 : WSTRING(94) := "Ratio apply to ramp signal to control Pvg Ev Tor when up axle oscillant movement is sollicited";
  gc_DbmTranslation_fr_Text1616 : WSTRING(27) := "Min pvg down axle oscillant";
  gc_DbmTranslation_fr_Text1617 : WSTRING(27) := "Max pvg down axle oscillant";
  gc_DbmTranslation_fr_Text1618 : WSTRING(96) := "Ratio apply to ramp signal to control Pvg Ev Tor when down axle oscillant movement is sollicited";
  gc_DbmTranslation_fr_Text1619 : WSTRING(96) := "Ratio apply to ramp signal to control Pvg Ev Tor when down axle oscillant movement is sollicited";
  gc_DbmTranslation_fr_Text1620 : WSTRING(96) := "Ratio apply to ramp signal to control Pvg Ev Tor when down axle oscillant movement is sollicited";
  gc_DbmTranslation_fr_Text1621 : WSTRING(20) := "Min pvg up axle fixe";
  gc_DbmTranslation_fr_Text1622 : WSTRING(20) := "Max pvg up axle fixe";
  gc_DbmTranslation_fr_Text1623 : WSTRING(89) := "Ratio apply to ramp signal to control Pvg Ev Tor when up axle fixe movement is sollicited";
  gc_DbmTranslation_fr_Text1624 : WSTRING(89) := "Ratio apply to ramp signal to control Pvg Ev Tor when up axle fixe movement is sollicited";
  gc_DbmTranslation_fr_Text1625 : WSTRING(89) := "Ratio apply to ramp signal to control Pvg Ev Tor when up axle fixe movement is sollicited";
  gc_DbmTranslation_fr_Text1626 : WSTRING(22) := "Min pvg down axle fixe";
  gc_DbmTranslation_fr_Text1627 : WSTRING(22) := "Max pvg down axle fixe";
  gc_DbmTranslation_fr_Text1628 : WSTRING(91) := "Ratio apply to ramp signal to control Pvg Ev Tor when down axle fixe movement is sollicited";
  gc_DbmTranslation_fr_Text1629 : WSTRING(91) := "Ratio apply to ramp signal to control Pvg Ev Tor when down axle fixe movement is sollicited";
  gc_DbmTranslation_fr_Text1630 : WSTRING(91) := "Ratio apply to ramp signal to control Pvg Ev Tor when down axle fixe movement is sollicited";
  gc_DbmTranslation_fr_Text1631 : WSTRING(97) := "Min pvg rotation counter clockwise basket with turret post in pourcent regarding batterie voltage";
  gc_DbmTranslation_fr_Text1632 : WSTRING(96) := "Max pvg rotation counter clockwise basket with Radio post in pourcent regarding batterie voltage";
  gc_DbmTranslation_fr_Text1633 : WSTRING(109) := "Ratio apply to ramp signal to control Pvg Ev Tor when rotation counter clockwise frame movement is sollicited";
  gc_DbmTranslation_fr_Text1634 : WSTRING(109) := "Ratio apply to ramp signal to control Pvg Ev Tor when rotation counter clockwise frame movement is sollicited";
  gc_DbmTranslation_fr_Text1635 : WSTRING(109) := "Ratio apply to ramp signal to control Pvg Ev Tor when rotation counter clockwise frame movement is sollicited";
  gc_DbmTranslation_fr_Text1636 : WSTRING(97) := "Min pvg rotation counter clockwise basket with turret post in pourcent regarding batterie voltage";
  gc_DbmTranslation_fr_Text1637 : WSTRING(96) := "Max pvg rotation counter clockwise basket with Radio post in pourcent regarding batterie voltage";
  gc_DbmTranslation_fr_Text1638 : WSTRING(109) := "Ratio apply to ramp signal to control Pvg Ev Tor when rotation counter clockwise frame movement is sollicited";
  gc_DbmTranslation_fr_Text1639 : WSTRING(109) := "Ratio apply to ramp signal to control Pvg Ev Tor when rotation counter clockwise frame movement is sollicited";
  gc_DbmTranslation_fr_Text1640 : WSTRING(109) := "Ratio apply to ramp signal to control Pvg Ev Tor when rotation counter clockwise frame movement is sollicited";
  gc_DbmTranslation_fr_Text1641 : WSTRING(42) := "Timer anti demarrage to detect start motor";
  gc_DbmTranslation_fr_Text1642 : WSTRING(45) := "Treshold rpm motor to control anti demarrage ";
  gc_DbmTranslation_fr_Text1643 : WSTRING(58) := "Slow speed apply to up delta arm when telescope is outside";
  gc_DbmTranslation_fr_Text1644 : WSTRING(60) := "Slow speed apply to down delta arm when telescope is outside";
  gc_DbmTranslation_fr_Text1645 : WSTRING(58) := "Slow speed apply to up arrow arm when telescope is outside";
  gc_DbmTranslation_fr_Text1646 : WSTRING(60) := "Slow speed apply to down arrow arm when telescope is outside";
  gc_DbmTranslation_fr_Text1647 : WSTRING(69) := "Slow speed apply to clockwise rotation turret when mode ALO is define";
  gc_DbmTranslation_fr_Text1648 : WSTRING(77) := "Slow speed apply to counter clockwise rotation turret when mode ALO is define";
  gc_DbmTranslation_fr_Text1649 : WSTRING(58) := "Slow speed apply to arrow arm down when mode ALO is define";
  gc_DbmTranslation_fr_Text1650 : WSTRING(79) := "Slow speed apply to rotation turret counter clockwise when telescope is outside";
  gc_DbmTranslation_fr_Text1651 : WSTRING(71) := "Slow speed apply to rotation turret clockwise when telescope is outside";
  gc_DbmTranslation_fr_Text1652 : WSTRING(62) := "Min pvg up mast measure in pourcent regarding batterie voltage";
  gc_DbmTranslation_fr_Text1653 : WSTRING(62) := "Max pvg up mast measure in pourcent regarding batterie voltage";
  gc_DbmTranslation_fr_Text1654 : WSTRING(25) := "Ramp time Up mast measure";
  gc_DbmTranslation_fr_Text1655 : WSTRING(25) := "Ramp time Up mast measure";
  gc_DbmTranslation_fr_Text1656 : WSTRING(25) := "Ramp time Up mast measure";
  gc_DbmTranslation_fr_Text1657 : WSTRING(64) := "Min pvg down mast measure in pourcent regarding batterie voltage";
  gc_DbmTranslation_fr_Text1658 : WSTRING(64) := "Max pvg down mast measure in pourcent regarding batterie voltage";
  gc_DbmTranslation_fr_Text1659 : WSTRING(27) := "Ramp time Down mast measure";
  gc_DbmTranslation_fr_Text1660 : WSTRING(27) := "Ramp time Down mast measure";
  gc_DbmTranslation_fr_Text1661 : WSTRING(27) := "Ramp time Down mast measure";
  gc_DbmTranslation_fr_Text1662 : WSTRING(62) := "Transmission1PressureSensor  - output characteristic - Positif";
  gc_DbmTranslation_fr_Text1663 : WSTRING(61) := "Transmission1PressureSensor - output characteristic - Neutral";
  gc_DbmTranslation_fr_Text1664 : WSTRING(61) := "Transmission1PressureSensor - output characteristic - Negatif";
  gc_DbmTranslation_fr_Text1665 : WSTRING(61) := "Transmission1PressureSensor  - input characteristic - Positif";
  gc_DbmTranslation_fr_Text1666 : WSTRING(60) := "Transmission1PressureSensor - input characteristic - Neutral";
  gc_DbmTranslation_fr_Text1667 : WSTRING(60) := "Transmission1PressureSensor - input characteristic - Negatif";
  gc_DbmTranslation_fr_Text1668 : WSTRING(62) := "Transmission2PressureSensor  - output characteristic - Positif";
  gc_DbmTranslation_fr_Text1669 : WSTRING(61) := "Transmission2PressureSensor - output characteristic - Neutral";
  gc_DbmTranslation_fr_Text1670 : WSTRING(61) := "Transmission2PressureSensor - output characteristic - Negatif";
  gc_DbmTranslation_fr_Text1671 : WSTRING(61) := "Transmission2PressureSensor  - input characteristic - Positif";
  gc_DbmTranslation_fr_Text1672 : WSTRING(60) := "Transmission2PressureSensor - input characteristic - Neutral";
  gc_DbmTranslation_fr_Text1673 : WSTRING(60) := "Transmission2PressureSensor - input characteristic - Negatif";
  gc_DbmTranslation_fr_Text1674 : WSTRING(54) := "BypassPressureSensor - output characteristic - Positif";
  gc_DbmTranslation_fr_Text1675 : WSTRING(54) := "BypassPressureSensor - output characteristic - Neutral";
  gc_DbmTranslation_fr_Text1676 : WSTRING(54) := "BypassPressureSensor - output characteristic - Negatif";
  gc_DbmTranslation_fr_Text1677 : WSTRING(53) := "BypassPressureSensor - input characteristic - Positif";
  gc_DbmTranslation_fr_Text1678 : WSTRING(53) := "BypassPressureSensor - input characteristic - Neutral";
  gc_DbmTranslation_fr_Text1679 : WSTRING(53) := "BypassPressureSensor - input characteristic - Negatif";
  gc_DbmTranslation_fr_Text1680 : WSTRING(18) := "Param debug Neotec";
  gc_DbmTranslation_fr_Text1681 : WSTRING(18) := "Param debug Neotec";
  gc_DbmTranslation_fr_Text1682 : WSTRING(18) := "Param debug Neotec";
  gc_DbmTranslation_fr_Text1683 : WSTRING(18) := "Param debug Neotec";
  gc_DbmTranslation_fr_Text1684 : WSTRING(18) := "Param debug Neotec";
  gc_DbmTranslation_fr_Text1685 : WSTRING(18) := "Param debug Neotec";
  gc_DbmTranslation_fr_Text1686 : WSTRING(18) := "Param debug Neotec";
  gc_DbmTranslation_fr_Text1687 : WSTRING(18) := "Param debug Neotec";
  gc_DbmTranslation_fr_Text1688 : WSTRING(18) := "Param debug Neotec";
  gc_DbmTranslation_fr_Text1689 : WSTRING(18) := "Param debug Neotec";
  gc_DbmTranslation_fr_Text1690 : WSTRING(18) := "Param debug Neotec";
  gc_DbmTranslation_fr_Text1691 : WSTRING(18) := "Param debug Neotec";
  gc_DbmTranslation_fr_Text1692 : WSTRING(18) := "Param debug Neotec";
  gc_DbmTranslation_fr_Text1693 : WSTRING(18) := "Param debug Neotec";
  gc_DbmTranslation_fr_Text1694 : WSTRING(18) := "Param debug Neotec";
  gc_DbmTranslation_fr_Text1695 : WSTRING(18) := "Param debug Neotec";
  gc_DbmTranslation_fr_Text1696 : WSTRING(18) := "Param debug Neotec";
  gc_DbmTranslation_fr_Text1697 : WSTRING(47) := "Current parameter for 220v appliqued on genetor";
  gc_DbmTranslation_fr_Text1698 : WSTRING(38) := "Number element of transission Pressure";
  gc_DbmTranslation_fr_Text1699 : WSTRING(20) := "Ramp up Ev Generator";
  gc_DbmTranslation_fr_Text1700 : WSTRING(20) := "Ramp Up Ev Generator";
  gc_DbmTranslation_fr_Text1701 : WSTRING(28) := "Gas gauge alarm min treshold";
  gc_DbmTranslation_fr_Text1702 : WSTRING(37) := "CRC of communication parameter SRDO 1";
  gc_DbmTranslation_fr_Text1703 : WSTRING(37) := "CRC of communication parameter SRDO 2";
  gc_DbmTranslation_fr_Text1704 : WSTRING(37) := "CRC of communication parameter SRDO 3";
  gc_DbmTranslation_fr_Text1705 : WSTRING(37) := "CRC of communication parameter SRDO 4";
  gc_DbmTranslation_fr_Text1706 : WSTRING(37) := "CRC of communication parameter SRDO 5";
  gc_DbmTranslation_fr_Text1707 : WSTRING(37) := "CRC of communication parameter SRDO 6";
  gc_DbmTranslation_fr_Text1708 : WSTRING(37) := "CRC of communication parameter SRDO 7";
  gc_DbmTranslation_fr_Text1709 : WSTRING(37) := "CRC of communication parameter SRDO 8";
  gc_DbmTranslation_fr_Text1710 : WSTRING(37) := "CRC of communication parameter SRDO 9";
  gc_DbmTranslation_fr_Text1711 : WSTRING(38) := "CRC of communication parameter SRDO 10";
  gc_DbmTranslation_fr_Text1712 : WSTRING(25) := "Timeout sdo resquest time";
  gc_DbmTranslation_fr_Text1713 : WSTRING(22) := "Activation des alarmes";
  gc_DbmTranslation_fr_Text1714 : WSTRING(32) := "Activation de l’alarme de bypass";
  gc_DbmTranslation_fr_Text1715 : WSTRING(68) := "TankOilTemperature - input current - output characteristic - Positif";
  gc_DbmTranslation_fr_Text1716 : WSTRING(68) := "TankOilTemperature - input current - output characteristic - Neutral";
  gc_DbmTranslation_fr_Text1717 : WSTRING(68) := "TankOilTemperature - input current - output characteristic - Negatif";
  gc_DbmTranslation_fr_Text1718 : WSTRING(65) := "Ratio apply to ramp signal to control arm delta with nacelle post";
  gc_DbmTranslation_fr_Text1719 : WSTRING(65) := "Ratio apply to ramp signal to control arm delta with nacelle post";
  gc_DbmTranslation_fr_Text1720 : WSTRING(65) := "Ratio apply to ramp signal to control arm delta with nacelle post";
  gc_DbmTranslation_fr_Text1721 : WSTRING(65) := "Ratio apply to ramp signal to control arm delta with nacelle post";
  gc_DbmTranslation_fr_Text1722 : WSTRING(65) := "Ratio apply to ramp signal to control arm delta with nacelle post";
  gc_DbmTranslation_fr_Text1723 : WSTRING(65) := "Ratio apply to ramp signal to control arm arrow with nacelle post";
  gc_DbmTranslation_fr_Text1724 : WSTRING(65) := "Ratio apply to ramp signal to control arm arrow with nacelle post";
  gc_DbmTranslation_fr_Text1725 : WSTRING(65) := "Ratio apply to ramp signal to control arm arrow with nacelle post";
  gc_DbmTranslation_fr_Text1726 : WSTRING(65) := "Ratio apply to ramp signal to control arm arrow with nacelle post";
  gc_DbmTranslation_fr_Text1727 : WSTRING(65) := "Ratio apply to ramp signal to control arm arrow with nacelle post";
  gc_DbmTranslation_fr_Text1728 : WSTRING(69) := "Ratio apply to ramp signal to control arm telescope with nacelle post";
  gc_DbmTranslation_fr_Text1729 : WSTRING(69) := "Ratio apply to ramp signal to control arm telescope with nacelle post";
  gc_DbmTranslation_fr_Text1730 : WSTRING(69) := "Ratio apply to ramp signal to control arm telescope with nacelle post";
  gc_DbmTranslation_fr_Text1731 : WSTRING(69) := "Ratio apply to ramp signal to control arm telescope with nacelle post";
  gc_DbmTranslation_fr_Text1732 : WSTRING(69) := "Ratio apply to ramp signal to control arm telescope with nacelle post";
  gc_DbmTranslation_fr_Text1733 : WSTRING(53) := "Ratio apply to ramp signal to control rotation turret";
  gc_DbmTranslation_fr_Text1734 : WSTRING(53) := "Ratio apply to ramp signal to control rotation turret";
  gc_DbmTranslation_fr_Text1735 : WSTRING(53) := "Ratio apply to ramp signal to control rotation turret";
  gc_DbmTranslation_fr_Text1736 : WSTRING(48) := "Ratio apply to ramp signal to control Pvg Ev Tor";
  gc_DbmTranslation_fr_Text1737 : WSTRING(48) := "Ratio apply to ramp signal to control Pvg Ev Tor";
  gc_DbmTranslation_fr_Text1738 : WSTRING(48) := "Ratio apply to ramp signal to control Pvg Ev Tor";
  gc_DbmTranslation_fr_Text1739 : WSTRING(48) := "Ratio apply to ramp signal to control Pvg Ev Tor";
  gc_DbmTranslation_fr_Text1740 : WSTRING(48) := "Ratio apply to ramp signal to control Pvg Ev Tor";
  gc_DbmTranslation_fr_Text1741 : WSTRING(40) := "Angle end stop low position of delta arm";
  gc_DbmTranslation_fr_Text1742 : WSTRING(63) := "Calibrate Angle end stop low position of delta arm master input";
  gc_DbmTranslation_fr_Text1743 : WSTRING(41) := "Angle end stop high position of delta arm";
  gc_DbmTranslation_fr_Text1744 : WSTRING(64) := "Calibrate Angle end stop high position of delta arm master input";
  gc_DbmTranslation_fr_Text1745 : WSTRING(40) := "Angle end stop low position of arrow arm";
  gc_DbmTranslation_fr_Text1746 : WSTRING(63) := "Calibrate Angle end stop low position of arrow arm master input";
  gc_DbmTranslation_fr_Text1747 : WSTRING(41) := "Angle end stop high position of arrow arm";
  gc_DbmTranslation_fr_Text1748 : WSTRING(64) := "Calibrate Angle end stop high position of arrow arm master input";
  gc_DbmTranslation_fr_Text1749 : WSTRING(31) := "Lenght end stop low telescope 1";
  gc_DbmTranslation_fr_Text1750 : WSTRING(32) := "Lenght end stop high telescope 1";
  gc_DbmTranslation_fr_Text1751 : WSTRING(41) := "Lenght calibrate end stop low telescope 1";
  gc_DbmTranslation_fr_Text1752 : WSTRING(43) := "Lenght calibrate  end stop high telescope 1";
  gc_DbmTranslation_fr_Text1753 : WSTRING(31) := "Lenght end stop low telescope 2";
  gc_DbmTranslation_fr_Text1754 : WSTRING(32) := "Lenght end stop high telescope 2";
  gc_DbmTranslation_fr_Text1755 : WSTRING(41) := "Lenght calibrate end stop low telescope 2";
  gc_DbmTranslation_fr_Text1756 : WSTRING(43) := "Lenght calibrate  end stop high telescope 2";
  gc_DbmTranslation_fr_Text1757 : WSTRING(64) := "Ratio apply to ramp signal to control arm delta with turret post";
  gc_DbmTranslation_fr_Text1758 : WSTRING(64) := "Ratio apply to ramp signal to control arm delta with turret post";
  gc_DbmTranslation_fr_Text1759 : WSTRING(64) := "Ratio apply to ramp signal to control arm delta with turret post";
  gc_DbmTranslation_fr_Text1760 : WSTRING(64) := "Ratio apply to ramp signal to control arm delta with turret post";
  gc_DbmTranslation_fr_Text1761 : WSTRING(64) := "Ratio apply to ramp signal to control arm delta with turret post";
  gc_DbmTranslation_fr_Text1762 : WSTRING(64) := "Ratio apply to ramp signal to control arm arrow with turret post";
  gc_DbmTranslation_fr_Text1763 : WSTRING(64) := "Ratio apply to ramp signal to control arm arrow with turret post";
  gc_DbmTranslation_fr_Text1764 : WSTRING(64) := "Ratio apply to ramp signal to control arm arrow with turret post";
  gc_DbmTranslation_fr_Text1765 : WSTRING(64) := "Ratio apply to ramp signal to control arm arrow with turret post";
  gc_DbmTranslation_fr_Text1766 : WSTRING(64) := "Ratio apply to ramp signal to control arm arrow with turret post";
  gc_DbmTranslation_fr_Text1767 : WSTRING(68) := "Ratio apply to ramp signal to control arm telescope with turret post";
  gc_DbmTranslation_fr_Text1768 : WSTRING(68) := "Ratio apply to ramp signal to control arm telescope with turret post";
  gc_DbmTranslation_fr_Text1769 : WSTRING(68) := "Ratio apply to ramp signal to control arm telescope with turret post";
  gc_DbmTranslation_fr_Text1770 : WSTRING(68) := "Ratio apply to ramp signal to control arm telescope with turret post";
  gc_DbmTranslation_fr_Text1771 : WSTRING(68) := "Ratio apply to ramp signal to control arm telescope with turret post";
  gc_DbmTranslation_fr_Text1772 : WSTRING(26) := "Angle calib delta arm hyst";
  gc_DbmTranslation_fr_Text1773 : WSTRING(26) := "Angle calib arrow arm hyst";
  gc_DbmTranslation_fr_Text1774 : WSTRING(63) := "Calibrate Angle end stop high position of delta arm slave input";
  gc_DbmTranslation_fr_Text1775 : WSTRING(62) := "Calibrate Angle end stop low position of delta arm slave input";
  gc_DbmTranslation_fr_Text1776 : WSTRING(64) := "Calibrate Angle end stop high position of arrow arm master input";
  gc_DbmTranslation_fr_Text1777 : WSTRING(63) := "Calibrate Angle end stop Low position of arrow arm master input";
  gc_DbmTranslation_fr_Text1778 : WSTRING(29) := "Up  Inclinaison basket button";
  gc_DbmTranslation_fr_Text1779 : WSTRING(40) := "Up  Inclinaison basket  button raw value";
  gc_DbmTranslation_fr_Text1780 : WSTRING(31) := "Down  Inclinaison basket button";
  gc_DbmTranslation_fr_Text1781 : WSTRING(41) := "Down  Inclinaison basket button raw value";
  gc_DbmTranslation_fr_Text1782 : WSTRING(18) := "Up pendular button";
  gc_DbmTranslation_fr_Text1783 : WSTRING(28) := "Up pendular button raw value";
  gc_DbmTranslation_fr_Text1784 : WSTRING(20) := "Down pendular button";
  gc_DbmTranslation_fr_Text1785 : WSTRING(30) := "Down pendular button raw value";
  gc_DbmTranslation_fr_Text1786 : WSTRING(40) := "Counter Clockwise rotation basket button";
  gc_DbmTranslation_fr_Text1787 : WSTRING(50) := "Counter Clockwise rotation basket button raw value";
  gc_DbmTranslation_fr_Text1788 : WSTRING(32) := "Clockwise rotation basket button";
  gc_DbmTranslation_fr_Text1789 : WSTRING(42) := "Clockwise rotation basket button raw value";
  gc_DbmTranslation_fr_Text1790 : WSTRING(10) := "Overload 1";
  gc_DbmTranslation_fr_Text1791 : WSTRING(20) := "Overload 1 raw value";
  gc_DbmTranslation_fr_Text1792 : WSTRING(10) := "Overload 2";
  gc_DbmTranslation_fr_Text1793 : WSTRING(20) := "Overload 2 raw value";
  gc_DbmTranslation_fr_Text1794 : WSTRING(34) := "Nacelle basket right side sensor 1";
  gc_DbmTranslation_fr_Text1795 : WSTRING(40) := "Nacelle basket right side sensor 1 value";
  gc_DbmTranslation_fr_Text1796 : WSTRING(40) := "Nacelle basket right side sensor 2 value";
  gc_DbmTranslation_fr_Text1797 : WSTRING(40) := "Nacelle basket right side sensor 2 value";
  gc_DbmTranslation_fr_Text1798 : WSTRING(33) := "Nacelle basket left side sensor 1";
  gc_DbmTranslation_fr_Text1799 : WSTRING(39) := "Nacelle basket left side sensor 1 value";
  gc_DbmTranslation_fr_Text1800 : WSTRING(33) := "Nacelle basket left side sensor 2";
  gc_DbmTranslation_fr_Text1801 : WSTRING(39) := "Nacelle basket left side sensor 2 value";
  gc_DbmTranslation_fr_Text1802 : WSTRING(26) := "Low sector pendular sensor";
  gc_DbmTranslation_fr_Text1803 : WSTRING(32) := "Low sector pendular sensor value";
  gc_DbmTranslation_fr_Text1804 : WSTRING(24) := "High Sector Plate Sensor";
  gc_DbmTranslation_fr_Text1805 : WSTRING(30) := "High Sector Plate Sensor value";
  gc_DbmTranslation_fr_Text1806 : WSTRING(20) := "Folded ladder sensor";
  gc_DbmTranslation_fr_Text1807 : WSTRING(26) := "Folded ladder sensor value";
  gc_DbmTranslation_fr_Text1808 : WSTRING(23) := "Safety man system value";
  gc_DbmTranslation_fr_Text1809 : WSTRING(29) := "Delta arm axis joystick value";
  gc_DbmTranslation_fr_Text1810 : WSTRING(29) := "Arrow arm axis joystick value";
  gc_DbmTranslation_fr_Text1811 : WSTRING(33) := "Telescope arm axis joystick value";
  gc_DbmTranslation_fr_Text1812 : WSTRING(35) := "Rotation turret axis joystick value";
  gc_DbmTranslation_fr_Text1813 : WSTRING(27) := "Advance axis joystick value";
  gc_DbmTranslation_fr_Text1814 : WSTRING(28) := "Rearmement Safety Man System";
  gc_DbmTranslation_fr_Text1815 : WSTRING(34) := "Rearmement Safety Man System value";
  gc_DbmTranslation_fr_Text1816 : WSTRING(28) := "Abutement Nacelle Track Side";
  gc_DbmTranslation_fr_Text1817 : WSTRING(34) := "Abutement Nacelle Track Side value";
  gc_DbmTranslation_fr_Text1818 : WSTRING(31) := "Abutement Nacelle Centered Side";
  gc_DbmTranslation_fr_Text1819 : WSTRING(37) := "Abutement Nacelle Centered Side value";
  gc_DbmTranslation_fr_Text1820 : WSTRING(24) := "Delta arm Joystick value";
  gc_DbmTranslation_fr_Text1821 : WSTRING(38) := "Arrow Joystick / centered turret value";
  gc_DbmTranslation_fr_Text1822 : WSTRING(31) := "Centered advance joystick value";
  gc_DbmTranslation_fr_Text1823 : WSTRING(20) := "Dead man pedal value";
  gc_DbmTranslation_fr_Text1824 : WSTRING(35) := "Pressence in nacelle sensor 1 value";
  gc_DbmTranslation_fr_Text1825 : WSTRING(35) := "Pressence in nacelle sensor 2 value";
  gc_DbmTranslation_fr_Text1826 : WSTRING(14) := "Gachette value";
  gc_DbmTranslation_fr_Text1827 : WSTRING(12) := "Klaxon value";
  gc_DbmTranslation_fr_Text1828 : WSTRING(17) := "Stop Motor button";
  gc_DbmTranslation_fr_Text1829 : WSTRING(28) := "Authorization work key value";
  gc_DbmTranslation_fr_Text1830 : WSTRING(27) := "Etallonnage Joystick Button";
  gc_DbmTranslation_fr_Text1831 : WSTRING(22) := "Close Portillon Sensor";
  gc_DbmTranslation_fr_Text1832 : WSTRING(31) := "Heartbeat for slave module 48xs";
  gc_DbmTranslation_fr_Text1833 : WSTRING(37) := "Batterie voltage of module slave 48xs";
  gc_DbmTranslation_fr_Text1834 : WSTRING(24) := "Rotation frame clockwise";
  gc_DbmTranslation_fr_Text1835 : WSTRING(32) := "Rotation frame Counter clockwise";
  gc_DbmTranslation_fr_Text1836 : WSTRING(40) := "Up pendular or rotation clockwise turret";
  gc_DbmTranslation_fr_Text1837 : WSTRING(50) := "down pendular or rotation counter clockwise turret";
  gc_DbmTranslation_fr_Text1838 : WSTRING(17) := "Selector pendular";
  gc_DbmTranslation_fr_Text1839 : WSTRING(24) := "Selector rotation turret";
  gc_DbmTranslation_fr_Text1840 : WSTRING(17) := "Up axle oscillant";
  gc_DbmTranslation_fr_Text1841 : WSTRING(19) := "Down axle oscillant";
  gc_DbmTranslation_fr_Text1842 : WSTRING(12) := "Up axle fixe";
  gc_DbmTranslation_fr_Text1843 : WSTRING(14) := "Down axle fixe";
  gc_DbmTranslation_fr_Text1844 : WSTRING(21) := "Forcing advance track";
  gc_DbmTranslation_fr_Text1845 : WSTRING(21) := "Autorize up delta arm";
  gc_DbmTranslation_fr_Text1846 : WSTRING(23) := "Autorize down delta arm";
  gc_DbmTranslation_fr_Text1847 : WSTRING(21) := "Autorize up arrow arm";
  gc_DbmTranslation_fr_Text1848 : WSTRING(23) := "Autorize down arrow arm";
  gc_DbmTranslation_fr_Text1849 : WSTRING(26) := "Autorize Out telescope arm";
  gc_DbmTranslation_fr_Text1850 : WSTRING(25) := "Autorize In telescope arm";
  gc_DbmTranslation_fr_Text1851 : WSTRING(34) := "Autorize rotation basket clockwise";
  gc_DbmTranslation_fr_Text1852 : WSTRING(42) := "Autorize rotation basket counter clockwise";
  gc_DbmTranslation_fr_Text1853 : WSTRING(30) := "Autorize up inclinaison basket";
  gc_DbmTranslation_fr_Text1854 : WSTRING(32) := "Autorize down inclinaison basket";
  gc_DbmTranslation_fr_Text1855 : WSTRING(20) := "Autorize up pendular";
  gc_DbmTranslation_fr_Text1856 : WSTRING(22) := "Autorize down pendular";
  gc_DbmTranslation_fr_Text1857 : WSTRING(34) := "Autorize rotation turret clockwise";
  gc_DbmTranslation_fr_Text1858 : WSTRING(42) := "Autorize rotation turret counter clockwise";
  gc_DbmTranslation_fr_Text1859 : WSTRING(17) := "Start Up current ";
  gc_DbmTranslation_fr_Text1860 : WSTRING(50) := "High forcing current when preheating is sollicited";
  gc_DbmTranslation_fr_Text1861 : WSTRING(19) := "Low forcing current";
  gc_DbmTranslation_fr_Text1862 : WSTRING(61) := "Threshold3 aplly when more at one Pvg movement are sollicited";
  gc_DbmTranslation_fr_Text1863 : WSTRING(52) := "Threshold2 aplly when one Pvg movement is sollicited";
  gc_DbmTranslation_fr_Text1864 : WSTRING(51) := "Threshold1 aplly when a movement on groupe2 output ";
  gc_DbmTranslation_fr_Text1865 : WSTRING(35) := "Time to pilot motor  while start up";
  gc_DbmTranslation_fr_Text1866 : WSTRING(38) := "Time to pilot motor  while preheating ";
  gc_DbmTranslation_fr_Text1867 : WSTRING(53) := "Current applu when Translation movement is sollicited";
  gc_DbmTranslation_fr_Text1868 : WSTRING(30) := "Current apply when no movement";
  gc_DbmTranslation_fr_Text1869 : WSTRING(25) := "Treshold regime generator";
  gc_DbmTranslation_fr_Text1870 : WSTRING(23) := "Engine Idle Speed Motor";
  gc_DbmTranslation_fr_Text1871 : WSTRING(45) := "Counter for filtred the no mouvement function";
  gc_DbmTranslation_fr_Text1872 : WSTRING(41) := "Error status of Motor Default Light ouput";
  gc_DbmTranslation_fr_Text1873 : WSTRING(19) := "Motor default light";
  gc_DbmTranslation_fr_Text1874 : WSTRING(36) := "Error status of Overload Light ouput";
  gc_DbmTranslation_fr_Text1875 : WSTRING(14) := "Overload Light";
  gc_DbmTranslation_fr_Text1876 : WSTRING(28) := "Error status of Buzzer ouput";
  gc_DbmTranslation_fr_Text1877 : WSTRING(6) := "Buzzer";
  gc_DbmTranslation_fr_Text1878 : WSTRING(35) := "Supply Dead Man Pedal and Joysticks";
  gc_DbmTranslation_fr_Text1879 : WSTRING(35) := "Error status of Warming Light ouput";
  gc_DbmTranslation_fr_Text1880 : WSTRING(13) := "Warming Light";
  gc_DbmTranslation_fr_Text1881 : WSTRING(42) := "Error status of devers default light ouput";
  gc_DbmTranslation_fr_Text1882 : WSTRING(20) := "Devers Default Light";
  gc_DbmTranslation_fr_Text1883 : WSTRING(35) := "Error status of Gas Oil Light ouput";
  gc_DbmTranslation_fr_Text1884 : WSTRING(12) := "GasOil Light";
  gc_DbmTranslation_fr_Text1885 : WSTRING(35) := "White light ARG basket error status";
  gc_DbmTranslation_fr_Text1886 : WSTRING(30) := "White light ARG basket command";
  gc_DbmTranslation_fr_Text1887 : WSTRING(33) := "Red light ARG basket error status";
  gc_DbmTranslation_fr_Text1888 : WSTRING(20) := "Red light ARG basket";
  gc_DbmTranslation_fr_Text1889 : WSTRING(33) := "Red light ARD basket error status";
  gc_DbmTranslation_fr_Text1890 : WSTRING(28) := "Red light ARD basket command";
  gc_DbmTranslation_fr_Text1891 : WSTRING(35) := "White light ARD basket error status";
  gc_DbmTranslation_fr_Text1892 : WSTRING(30) := "White light ARD basket command";
  gc_DbmTranslation_fr_Text1893 : WSTRING(33) := "White light Ar 15746 error status";
  gc_DbmTranslation_fr_Text1894 : WSTRING(24) := "White light Ar 15746 cmd";
  gc_DbmTranslation_fr_Text1895 : WSTRING(25) := "Restriced mode aru active";
  gc_DbmTranslation_fr_Text1896 : WSTRING(54) := "Translation movement is solicited, info to pilot motor";
  gc_DbmTranslation_fr_Text1897 : WSTRING(26) := "Axle movement is solicited";
  gc_DbmTranslation_fr_Text1898 : WSTRING(21) := "Down axle fixe sensor";
  gc_DbmTranslation_fr_Text1899 : WSTRING(26) := "Down axle oscillant sensor";
  gc_DbmTranslation_fr_Text1900 : WSTRING(11) := "Slope Angle";
  gc_DbmTranslation_fr_Text1901 : WSTRING(49) := "Reduce the speed of the turret clockwise movement";
  gc_DbmTranslation_fr_Text1902 : WSTRING(57) := "Reduce the speed of the turret counter clockwise movement";
  gc_DbmTranslation_fr_Text1903 : WSTRING(47) := "Reduce the speed of the arrow arm down movement";
  gc_DbmTranslation_fr_Text1904 : WSTRING(34) := "Stop the turret clockwise movement";
  gc_DbmTranslation_fr_Text1905 : WSTRING(42) := "Stop the turret counter clockwise movement";
  gc_DbmTranslation_fr_Text1906 : WSTRING(34) := "Stop the basket clockwise movement";
  gc_DbmTranslation_fr_Text1907 : WSTRING(42) := "Stop the basket counter clockwise movement";
  gc_DbmTranslation_fr_Text1908 : WSTRING(32) := "Stop the arrow arm down movement";
  gc_DbmTranslation_fr_Text1909 : WSTRING(31) := "Stop the telescope out movement";
  gc_DbmTranslation_fr_Text1910 : WSTRING(23) := "Encodeur turret 1 angle";
  gc_DbmTranslation_fr_Text1911 : WSTRING(28) := "Red light ARG basket command";
  gc_DbmTranslation_fr_Text1912 : WSTRING(30) := "White light ARG basket command";
  gc_DbmTranslation_fr_Text1913 : WSTRING(38) := "Encodeur mast measure raw value sensor";
  gc_DbmTranslation_fr_Text1914 : WSTRING(22) := "Worg abutments and key";
  gc_DbmTranslation_fr_Text1915 : WSTRING(20) := "Speed vehicle in kmh";
  gc_DbmTranslation_fr_Text1916 : WSTRING(46) := "Stop all movement when a test brake is running";
  gc_DbmTranslation_fr_Text1917 : WSTRING(50) := "Stop all movement when a break in brake is running";
  gc_DbmTranslation_fr_Text1918 : WSTRING(37) := "Enable buzzer by select post function";
  gc_DbmTranslation_fr_Text1919 : WSTRING(19) := "Select control Post";
  gc_DbmTranslation_fr_Text1920 : WSTRING(21) := "Centered Turret state";
  gc_DbmTranslation_fr_Text1921 : WSTRING(14) := "Authorize Work";
  gc_DbmTranslation_fr_Text1922 : WSTRING(26) := "Up osccilant axle position";
  gc_DbmTranslation_fr_Text1923 : WSTRING(21) := "Up fixe axle position";
  gc_DbmTranslation_fr_Text1924 : WSTRING(14) := "Rail word mode";
  gc_DbmTranslation_fr_Text1925 : WSTRING(18) := "Ev forward command";
  gc_DbmTranslation_fr_Text1926 : WSTRING(19) := "Ev backward command";
  gc_DbmTranslation_fr_Text1927 : WSTRING(28) := "Red light ARD basket command";
  gc_DbmTranslation_fr_Text1928 : WSTRING(30) := "White light ARD basket command";
  gc_DbmTranslation_fr_Text1929 : WSTRING(24) := "Second Park Brake Active";
  gc_DbmTranslation_fr_Text1930 : WSTRING(33) := "Autorisation High Speed Key State";
  gc_DbmTranslation_fr_Text1931 : WSTRING(46) := "Translation on Rail with Electric Ramp Ongoing";
  gc_DbmTranslation_fr_Text1932 : WSTRING(18) := "Rpm Pvg Trans Rail";
  gc_DbmTranslation_fr_Text1933 : WSTRING(11) := "Battery Soc";
  gc_DbmTranslation_fr_Text1934 : WSTRING(15) := "Current Battery";
  gc_DbmTranslation_fr_Text1935 : WSTRING(29) := "Send Authorize Reload Battery";
  gc_DbmTranslation_fr_Text1936 : WSTRING(14) := "Battery Status";
  gc_DbmTranslation_fr_Text1937 : WSTRING(14) := "Preheat Status";
  gc_DbmTranslation_fr_Text1938 : WSTRING(22) := "Engine Faillure Status";
  gc_DbmTranslation_fr_Text1939 : WSTRING(18) := "Maintenance Status";
  gc_DbmTranslation_fr_Text1940 : WSTRING(10) := "Oil Status";
  gc_DbmTranslation_fr_Text1941 : WSTRING(21) := "Delta Arm Sector Down";
  gc_DbmTranslation_fr_Text1942 : WSTRING(21) := "Arrow Arm Sector Down";
  gc_DbmTranslation_fr_Text1943 : WSTRING(20) := "Pendular Sector Down";
  gc_DbmTranslation_fr_Text1944 : WSTRING(19) := "Delta Arm in Center";
  gc_DbmTranslation_fr_Text1945 : WSTRING(19) := "Arrow Arm in Center";
  gc_DbmTranslation_fr_Text1946 : WSTRING(18) := "Pendular in Center";
  gc_DbmTranslation_fr_Text1947 : WSTRING(25) := "Basket Rotation in Center";
  gc_DbmTranslation_fr_Text1948 : WSTRING(19) := "Telescope in Center";
  gc_DbmTranslation_fr_Text1949 : WSTRING(28) := "Basket Inclinaison in Center";
  gc_DbmTranslation_fr_Text1950 : WSTRING(25) := "Delta Arm Move Up Allowed";
  gc_DbmTranslation_fr_Text1951 : WSTRING(27) := "Delta Arm Move Down Allowed";
  gc_DbmTranslation_fr_Text1952 : WSTRING(25) := "Arrow Arm Move Up Allowed";
  gc_DbmTranslation_fr_Text1953 : WSTRING(27) := "Arrow Arm Move Down Allowed";
  gc_DbmTranslation_fr_Text1954 : WSTRING(24) := "Pendular Move Up Allowed";
  gc_DbmTranslation_fr_Text1955 : WSTRING(26) := "Pendular Move Down Allowed";
  gc_DbmTranslation_fr_Text1956 : WSTRING(26) := "Telescope Move Out Allowed";
  gc_DbmTranslation_fr_Text1957 : WSTRING(25) := "Telescope Move In Allowed";
  gc_DbmTranslation_fr_Text1958 : WSTRING(37) := "Turret Counter Clockwise Move Allowed";
  gc_DbmTranslation_fr_Text1959 : WSTRING(29) := "Turret Clockwise Move Allowed";
  gc_DbmTranslation_fr_Text1960 : WSTRING(46) := "Basket Rotation Counter Clockwise Move Allowed";
  gc_DbmTranslation_fr_Text1961 : WSTRING(38) := "Basket Rotation Clockwise Move Allowed";
  gc_DbmTranslation_fr_Text1962 : WSTRING(34) := "Basket Inclinaison Move Up Allowed";
  gc_DbmTranslation_fr_Text1963 : WSTRING(36) := "Basket Inclinaison Move Down Allowed";
  gc_DbmTranslation_fr_Text1964 : WSTRING(25) := "Vehicule in Default (A12)";
  gc_DbmTranslation_fr_Text1965 : WSTRING(31) := "Telescope output possible (A48)";
  gc_DbmTranslation_fr_Text1966 : WSTRING(29) := "Telescope Winder Fault (A17) ";
  gc_DbmTranslation_fr_Text1967 : WSTRING(21) := "Nacelle post selector";
  gc_DbmTranslation_fr_Text1968 : WSTRING(11) := "STOP Status";
  gc_DbmTranslation_fr_Text1969 : WSTRING(18) := "SafeManSystem (A5)";
  gc_DbmTranslation_fr_Text1970 : WSTRING(22) := "High Speed Allow (A19)";
  gc_DbmTranslation_fr_Text1971 : WSTRING(43) := "Automatique Stop or function mismatch (A20)";
  gc_DbmTranslation_fr_Text1972 : WSTRING(24) := "Low Speed by fault (A46)";
  gc_DbmTranslation_fr_Text1973 : WSTRING(28) := "Measuring Mast in Fault (A8)";
  gc_DbmTranslation_fr_Text1974 : WSTRING(14) := "Fuel in Litter";
  gc_DbmTranslation_fr_Text1975 : WSTRING(20) := "Battery Voltage (Mv)";
  gc_DbmTranslation_fr_Text1976 : WSTRING(40) := "Train Transmission Pressure in Bar (A28)";
  gc_DbmTranslation_fr_Text1977 : WSTRING(33) := "Life byte sent to the controllers";
  gc_DbmTranslation_fr_Text1978 : WSTRING(35) := "Delta arm move up button is pressed";
  gc_DbmTranslation_fr_Text1979 : WSTRING(37) := "Delta arm move down button is pressed";
  gc_DbmTranslation_fr_Text1980 : WSTRING(35) := "Arrow arm move up button is pressed";
  gc_DbmTranslation_fr_Text1981 : WSTRING(37) := "Arrow arm move down button is pressed";
  gc_DbmTranslation_fr_Text1982 : WSTRING(34) := "Pendular move up button is pressed";
  gc_DbmTranslation_fr_Text1983 : WSTRING(36) := "Pendular move down button is pressed";
  gc_DbmTranslation_fr_Text1984 : WSTRING(36) := "Telescope move out button is pressed";
  gc_DbmTranslation_fr_Text1985 : WSTRING(35) := "Telescope move in button is pressed";
  gc_DbmTranslation_fr_Text1986 : WSTRING(44) := "Basket inclinaison move up button is pressed";
  gc_DbmTranslation_fr_Text1987 : WSTRING(46) := "Basket inclinaison move down button is pressed";
  gc_DbmTranslation_fr_Text1988 : WSTRING(41) := "Rotate turret clockwise button is pressed";
  gc_DbmTranslation_fr_Text1989 : WSTRING(49) := "Rotate turret counter clockwise button is pressed";
  gc_DbmTranslation_fr_Text1990 : WSTRING(41) := "Basket rotation move up button is pressed";
  gc_DbmTranslation_fr_Text1991 : WSTRING(43) := "Basket rotation move down button is pressed";
  gc_DbmTranslation_fr_Text1992 : WSTRING(23) := "Key RPM Selection level";
  gc_DbmTranslation_fr_Text1993 : WSTRING(32) := "Key Desactivation RPM selection ";
  gc_DbmTranslation_fr_Text1994 : WSTRING(51) := "Activation forcing White Rail lights Front and Rear";
  gc_DbmTranslation_fr_Text1995 : WSTRING(16) := "Activation neons";
  gc_DbmTranslation_fr_Text1996 : WSTRING(19) := "Key Calibration Min";
  gc_DbmTranslation_fr_Text1997 : WSTRING(19) := "Key Calibration Max";
  gc_DbmTranslation_fr_Text1998 : WSTRING(26) := "Key Calibration Validation";
  gc_DbmTranslation_fr_Text1999 : WSTRING(89) := "Element choice 1=Telescope; 2=Arrow arm; 3=Delta arm; 4=Turret; 5=Slope; 6=Measuring Mast";
  gc_DbmTranslation_fr_Text2000 : WSTRING(27) := "Key Calibration Max (-180°)";
  gc_DbmTranslation_fr_Text2001 : WSTRING(28) := "Key Slope Longitudinal reset";
  gc_DbmTranslation_fr_Text2002 : WSTRING(27) := "Key Slope Transversal reset";
  gc_DbmTranslation_fr_Text2003 : WSTRING(16) := "Active page opus";
  gc_DbmTranslation_fr_Text2004 : WSTRING(31) := "Key : YES reload with generator";
  gc_DbmTranslation_fr_Text2005 : WSTRING(30) := "Key : NO reload with generator";
  gc_DbmTranslation_fr_Text2006 : WSTRING(66) := "Command to perform the calibration of angle end stop low delta arm";
  gc_DbmTranslation_fr_Text2007 : WSTRING(67) := "Command to perform the calibration of angle end stop high delta arm";
  gc_DbmTranslation_fr_Text2008 : WSTRING(66) := "Command to perform the calibration of angle end stop low arrow arm";
  gc_DbmTranslation_fr_Text2009 : WSTRING(67) := "Command to perform the calibration of angle end stop high arrow arm";
  gc_DbmTranslation_fr_Text2010 : WSTRING(43) := "Command to savedcalibration value on EEPROM";
  gc_DbmTranslation_fr_Text2011 : WSTRING(71) := "Command to perform the calibration of lenght end stop low telescope arm";
  gc_DbmTranslation_fr_Text2012 : WSTRING(72) := "Command to perform the calibration of lenght end stop high telescope arm";
  gc_DbmTranslation_fr_Text2013 : WSTRING(39) := "Slope Telescope Mode Curve Slope Angles";
  gc_DbmTranslation_fr_Text2014 : WSTRING(39) := "Slope Telescope Mode Curve Slope Angles";
  gc_DbmTranslation_fr_Text2015 : WSTRING(39) := "Slope Telescope Mode Curve Slope Angles";
  gc_DbmTranslation_fr_Text2016 : WSTRING(39) := "Slope Telescope Mode Curve Slope Angles";
  gc_DbmTranslation_fr_Text2017 : WSTRING(39) := "Slope Telescope Mode Curve Slope Angles";
  gc_DbmTranslation_fr_Text2018 : WSTRING(39) := "Slope Telescope Mode Curve Slope Angles";
  gc_DbmTranslation_fr_Text2019 : WSTRING(39) := "Slope Telescope Mode Curve Slope Angles";
  gc_DbmTranslation_fr_Text2020 : WSTRING(39) := "Slope Telescope Mode Curve Slope Angles";
  gc_DbmTranslation_fr_Text2021 : WSTRING(39) := "Slope Telescope Mode Curve Slope Angles";
  gc_DbmTranslation_fr_Text2022 : WSTRING(39) := "Slope Telescope Mode Curve Slope Angles";
  gc_DbmTranslation_fr_Text2023 : WSTRING(44) := "Slope Telescope Mode Curve Telescope Lenghts";
  gc_DbmTranslation_fr_Text2024 : WSTRING(44) := "Slope Telescope Mode Curve Telescope Lenghts";
  gc_DbmTranslation_fr_Text2025 : WSTRING(44) := "Slope Telescope Mode Curve Telescope Lenghts";
  gc_DbmTranslation_fr_Text2026 : WSTRING(44) := "Slope Telescope Mode Curve Telescope Lenghts";
  gc_DbmTranslation_fr_Text2027 : WSTRING(44) := "Slope Telescope Mode Curve Telescope Lenghts";
  gc_DbmTranslation_fr_Text2028 : WSTRING(44) := "Slope Telescope Mode Curve Telescope Lenghts";
  gc_DbmTranslation_fr_Text2029 : WSTRING(44) := "Slope Telescope Mode Curve Telescope Lenghts";
  gc_DbmTranslation_fr_Text2030 : WSTRING(44) := "Slope Telescope Mode Curve Telescope Lenghts";
  gc_DbmTranslation_fr_Text2031 : WSTRING(44) := "Slope Telescope Mode Curve Telescope Lenghts";
  gc_DbmTranslation_fr_Text2032 : WSTRING(44) := "Slope Telescope Mode Curve Telescope Lenghts";
  gc_DbmTranslation_fr_Text2033 : WSTRING(106) := "Telescope limitation, threshold of the critical zone (relative to the stroke threshold given by the curve)";
  gc_DbmTranslation_fr_Text2034 : WSTRING(82) := "Telescope limitation, hysteresis applied on the critical zone threshold (relative)";
  gc_DbmTranslation_fr_Text2035 : WSTRING(66) := "Delta arm limitation, threshold use to detect if the slope is high";
  gc_DbmTranslation_fr_Text2036 : WSTRING(79) := "Delta arm limitation, hysteresis applied on the slope high threshold (relative)";
  gc_DbmTranslation_fr_Text2037 : WSTRING(66) := "Delta arm limitation, threshold angle of the upper zone (absolute)";
  gc_DbmTranslation_fr_Text2038 : WSTRING(79) := "Delta arm limitation, hysteresis applied on the upper zone threshold (relative)";
  gc_DbmTranslation_fr_Text2039 : WSTRING(98) := "Delta arm limitation, threshold angle of the slow down zone (relative to the upper zone threshold)";
  gc_DbmTranslation_fr_Text2040 : WSTRING(82) := "Delta arm limitation, extra speed reduction applied on slow speed (in perthousand)";
  gc_DbmTranslation_fr_Text2041 : WSTRING(97) := "Delta arm limitation, threshold angle of the critical zone (relative to the upper zone threshold)";
  gc_DbmTranslation_fr_Text2042 : WSTRING(82) := "Delta arm limitation, hysteresis applied on the critical zone threshold (relative)";
  gc_DbmTranslation_fr_Text2043 : WSTRING(66) := "Arrow arm limitation, threshold angle of the lower zone (absolute)";
  gc_DbmTranslation_fr_Text2044 : WSTRING(79) := "Arrow arm limitation, hysteresis applied on the lower zone threshold (relative)";
  gc_DbmTranslation_fr_Text2045 : WSTRING(98) := "Arrow arm limitation, threshold angle of the slow down zone (relative to the lower zone threshold)";
  gc_DbmTranslation_fr_Text2046 : WSTRING(82) := "Arrow arm limitation, extra speed reduction applied on slow speed (in perthousand)";
  gc_DbmTranslation_fr_Text2047 : WSTRING(97) := "Arrow arm limitation, threshold angle of the critical zone (relative to the lower zone threshold)";
  gc_DbmTranslation_fr_Text2048 : WSTRING(82) := "Arrow arm limitation, hysteresis applied on the critical zone threshold (relative)";
  gc_DbmTranslation_fr_Text2049 : WSTRING(35) := "Arm telescope mode curve arm angles";
  gc_DbmTranslation_fr_Text2050 : WSTRING(35) := "Arm telescope mode curve arm angles";
  gc_DbmTranslation_fr_Text2051 : WSTRING(35) := "Arm telescope mode curve arm angles";
  gc_DbmTranslation_fr_Text2052 : WSTRING(35) := "Arm telescope mode curve arm angles";
  gc_DbmTranslation_fr_Text2053 : WSTRING(35) := "Arm telescope mode curve arm angles";
  gc_DbmTranslation_fr_Text2054 : WSTRING(35) := "Arm telescope mode curve arm angles";
  gc_DbmTranslation_fr_Text2055 : WSTRING(35) := "Arm telescope mode curve arm angles";
  gc_DbmTranslation_fr_Text2056 : WSTRING(35) := "Arm telescope mode curve arm angles";
  gc_DbmTranslation_fr_Text2057 : WSTRING(35) := "Arm telescope mode curve arm angles";
  gc_DbmTranslation_fr_Text2058 : WSTRING(35) := "Arm telescope mode curve arm angles";
  gc_DbmTranslation_fr_Text2059 : WSTRING(41) := "Arm Telescope Mode Curve Telescopes Lengt";
  gc_DbmTranslation_fr_Text2060 : WSTRING(41) := "Arm Telescope Mode Curve Telescopes Lengt";
  gc_DbmTranslation_fr_Text2061 : WSTRING(41) := "Arm Telescope Mode Curve Telescopes Lengt";
  gc_DbmTranslation_fr_Text2062 : WSTRING(41) := "Arm Telescope Mode Curve Telescopes Lengt";
  gc_DbmTranslation_fr_Text2063 : WSTRING(41) := "Arm Telescope Mode Curve Telescopes Lengt";
  gc_DbmTranslation_fr_Text2064 : WSTRING(41) := "Arm Telescope Mode Curve Telescopes Lengt";
  gc_DbmTranslation_fr_Text2065 : WSTRING(41) := "Arm Telescope Mode Curve Telescopes Lengt";
  gc_DbmTranslation_fr_Text2066 : WSTRING(41) := "Arm Telescope Mode Curve Telescopes Lengt";
  gc_DbmTranslation_fr_Text2067 : WSTRING(41) := "Arm Telescope Mode Curve Telescopes Lengt";
  gc_DbmTranslation_fr_Text2068 : WSTRING(41) := "Arm Telescope Mode Curve Telescopes Lengt";
  gc_DbmTranslation_fr_Text2069 : WSTRING(20) := "Slope telescope mode";
  gc_DbmTranslation_fr_Text2070 : WSTRING(54) := "Thres of the high sector of Arrow for the STRUKTON EVO";
  gc_DbmTranslation_fr_Text2071 : WSTRING(53) := "Thres of the low sector of Arrow for the STRUKTON EVO";
  gc_DbmTranslation_fr_Text2072 : WSTRING(41) := "Hyst of sector Arrow for the STRUKTON EVO";
  gc_DbmTranslation_fr_Text2073 : WSTRING(41) := "Reduce the speed of the delta up movement";
  gc_DbmTranslation_fr_Text2074 : WSTRING(47) := "Reduce the speed of the arrow arm down movement";
  gc_DbmTranslation_fr_Text2075 : WSTRING(31) := "Stop the telescope out movement";
  gc_DbmTranslation_fr_Text2076 : WSTRING(30) := "Stop the delta arm up movement";
  gc_DbmTranslation_fr_Text2077 : WSTRING(32) := "Stop the arrow arm down movement";
  gc_DbmTranslation_fr_Text2078 : WSTRING(51) := "Stop all movement (a critical position was reached)";
  gc_DbmTranslation_fr_Text2079 : WSTRING(26) := "Selected slope angle value";
  gc_DbmTranslation_fr_Text2080 : WSTRING(71) := "Telescope limitation, stroke threshold extracted from the look up table";
  gc_DbmTranslation_fr_Text2081 : WSTRING(37) := "The telescope is in the critical zone";
  gc_DbmTranslation_fr_Text2082 : WSTRING(17) := "The slope is high";
  gc_DbmTranslation_fr_Text2083 : WSTRING(34) := "The delta arm is in the upper zone";
  gc_DbmTranslation_fr_Text2084 : WSTRING(37) := "The delta arm is in the critical zone";
  gc_DbmTranslation_fr_Text2085 : WSTRING(34) := "The arrow arm is in the lower zone";
  gc_DbmTranslation_fr_Text2086 : WSTRING(37) := "The arrow arm is in the critical zone";
  gc_DbmTranslation_fr_Text2087 : WSTRING(80) := "Enable simulation mode (use the simulation variables instead of the real inputs)";
  gc_DbmTranslation_fr_Text2088 : WSTRING(60) := "Variable used to simulate the longitudinal slope angle input";
  gc_DbmTranslation_fr_Text2089 : WSTRING(59) := "Variable used to simulate the transversal slope angle input";
  gc_DbmTranslation_fr_Text2090 : WSTRING(54) := "Variable used to simulate the telescope position input";
  gc_DbmTranslation_fr_Text2091 : WSTRING(60) := "Variable used to simulate the delta arm angular sensor input";
  gc_DbmTranslation_fr_Text2092 : WSTRING(60) := "Variable used to simulate the arrow arm angular sensor input";
  gc_DbmTranslation_fr_Text2093 : WSTRING(33) := "State heart beat telescope sensor";
  gc_DbmTranslation_fr_Text2094 : WSTRING(18) := "Lenght telescope 1";
  gc_DbmTranslation_fr_Text2095 : WSTRING(37) := "Error number of retractor telescope 1";
  gc_DbmTranslation_fr_Text2096 : WSTRING(27) := "Retractor Telescope value 1";
  gc_DbmTranslation_fr_Text2097 : WSTRING(18) := "Lenght telescope 2";
  gc_DbmTranslation_fr_Text2098 : WSTRING(37) := "Error number of retractor telescope 2";
  gc_DbmTranslation_fr_Text2099 : WSTRING(27) := "Retractor Telescope value 2";
  gc_DbmTranslation_fr_Text2100 : WSTRING(45) := "Reduce speed of the turret clockwise movement";
  gc_DbmTranslation_fr_Text2101 : WSTRING(34) := "Stop the turret clockwise movement";
  gc_DbmTranslation_fr_Text2102 : WSTRING(53) := "Reduce speed of the turret counter clockwise movement";
  gc_DbmTranslation_fr_Text2103 : WSTRING(42) := "Stop the turret counter clockwise movement";
  gc_DbmTranslation_fr_Text2104 : WSTRING(43) := "Reduce speed of the delta arm down movement";
  gc_DbmTranslation_fr_Text2105 : WSTRING(16) := "Folded delta arm";
  gc_DbmTranslation_fr_Text2106 : WSTRING(41) := "Reduce speed of the delta arm up movement";
  gc_DbmTranslation_fr_Text2107 : WSTRING(29) := "Test variable turret position";
  gc_DbmTranslation_fr_Text2108 : WSTRING(32) := "Test variable delta arm position";
  gc_DbmTranslation_fr_Text2109 : WSTRING(16) := "Folded arrow arm";
  gc_DbmTranslation_fr_Text2110 : WSTRING(35) := "Active reduce speed of arrow arm up";
  gc_DbmTranslation_fr_Text2111 : WSTRING(37) := "Active reduce speed of arrow arm down";
  gc_DbmTranslation_fr_Text2112 : WSTRING(39) := "Active reduce speed of telescope folded";
  gc_DbmTranslation_fr_Text2113 : WSTRING(29) := "Reduce speed for Telescope Up";
  gc_DbmTranslation_fr_Text2114 : WSTRING(31) := "Reduce speed for Telescope Down";
  gc_DbmTranslation_fr_Text2115 : WSTRING(30) := "Telescope folded position Stop";
  gc_DbmTranslation_fr_Text2116 : WSTRING(40) := "Autorise translation with unfolded Arrow";
  gc_DbmTranslation_fr_Text2117 : WSTRING(32) := "Valid position for the Telescope";
  gc_DbmTranslation_fr_Text2118 : WSTRING(48) := "Valid position for the first sector of Telescope";
  gc_DbmTranslation_fr_Text2119 : WSTRING(34) := "Turret negative end stop threshold";
  gc_DbmTranslation_fr_Text2120 : WSTRING(56) := "Turret negative end stop threshold hysteresis (relative)";
  gc_DbmTranslation_fr_Text2121 : WSTRING(91) := "Turret negative end stop threshold use to reduce speed (relative to the end stop threshold)";
  gc_DbmTranslation_fr_Text2122 : WSTRING(34) := "Turret positive end stop threshold";
  gc_DbmTranslation_fr_Text2123 : WSTRING(56) := "Turret positive end stop threshold hysteresis (relative)";
  gc_DbmTranslation_fr_Text2124 : WSTRING(91) := "Turret positive end stop threshold use to reduce speed (relative to the end stop threshold)";
  gc_DbmTranslation_fr_Text2125 : WSTRING(32) := "Folded Delta arm angle threshold";
  gc_DbmTranslation_fr_Text2126 : WSTRING(48) := "Folded Delta arm threshold hysteresis (relative)";
  gc_DbmTranslation_fr_Text2127 : WSTRING(92) := "Delta arm bottom end stop threshold use to reduce speed (relative to the end stop threshold)";
  gc_DbmTranslation_fr_Text2128 : WSTRING(32) := "Delta arm top end stop threshold";
  gc_DbmTranslation_fr_Text2129 : WSTRING(54) := "Delta arm top end stop threshold hysteresis (relative)";
  gc_DbmTranslation_fr_Text2130 : WSTRING(89) := "Delta arm top end stop threshold use to reduce speed (relative to the end stop threshold)";
  gc_DbmTranslation_fr_Text2131 : WSTRING(32) := "Folded Delta arm angle threshold";
  gc_DbmTranslation_fr_Text2132 : WSTRING(57) := "Arrow arm bottom end stop threshold hysteresis (relative)";
  gc_DbmTranslation_fr_Text2133 : WSTRING(67) := "Down Delta arm slow speed reduc when delta arm is close at abutment";
  gc_DbmTranslation_fr_Text2134 : WSTRING(44) := "Arrow Arm at the Top End Stop Slow Threshold";
  gc_DbmTranslation_fr_Text2135 : WSTRING(40) := "Arrow Arm Bottom End Stop Slow Threshold";
  gc_DbmTranslation_fr_Text2136 : WSTRING(32) := "Arrow Arm Top End Stop Threshold";
  gc_DbmTranslation_fr_Text2137 : WSTRING(32) := "Arrow Arm Slow Mvt Down End Stop";
  gc_DbmTranslation_fr_Text2138 : WSTRING(30) := "Arrow Arm Slow Mvt Up End Stop";
  gc_DbmTranslation_fr_Text2139 : WSTRING(34) := "Telescope Slow Mvt Folded End Stop";
  gc_DbmTranslation_fr_Text2140 : WSTRING(33) := "Thres of maximum Telescope sector";
  gc_DbmTranslation_fr_Text2141 : WSTRING(40) := "Hyst of thres to the sector of Telescope";
  gc_DbmTranslation_fr_Text2142 : WSTRING(42) := "Thres for the slow sector to the Telescope";
  gc_DbmTranslation_fr_Text2143 : WSTRING(34) := "Rear center position of the turret";
  gc_DbmTranslation_fr_Text2144 : WSTRING(61) := "Front center position of the turret in the positive direction";
  gc_DbmTranslation_fr_Text2145 : WSTRING(61) := "Front center position of the turret in the negative direction";
  gc_DbmTranslation_fr_Text2146 : WSTRING(60) := "Turret center zone window (relative to the center positions)";
  gc_DbmTranslation_fr_Text2147 : WSTRING(62) := "Hysteresis applied to the turret center zone window (relative)";
  gc_DbmTranslation_fr_Text2148 : WSTRING(93) := "Threshold use to reduce speed before reaching a center zone (relative to the center position)";
  gc_DbmTranslation_fr_Text2149 : WSTRING(66) := "Turret center zone window left  (relative to the center positions)";
  gc_DbmTranslation_fr_Text2150 : WSTRING(66) := "Turret center zone window right (relative to the center positions)";
  gc_DbmTranslation_fr_Text2151 : WSTRING(33) := "Stop the basket rotation movement";
  gc_DbmTranslation_fr_Text2152 : WSTRING(33) := "Stop the turret rotation movement";
  gc_DbmTranslation_fr_Text2153 : WSTRING(49) := "Reduce the speed of the turret clockwise movement";
  gc_DbmTranslation_fr_Text2154 : WSTRING(57) := "Reduce the speed of the turret counter clockwise movement";
  gc_DbmTranslation_fr_Text2155 : WSTRING(30) := "Turret is in a center position";
  gc_DbmTranslation_fr_Text2156 : WSTRING(80) := "Enable simulation mode (use the simulation variables instead of the real inputs)";
  gc_DbmTranslation_fr_Text2157 : WSTRING(54) := "Test variable for simulation - basket left side sensor";
  gc_DbmTranslation_fr_Text2158 : WSTRING(55) := "Test variable for simulation - basket right side sensor";
  gc_DbmTranslation_fr_Text2159 : WSTRING(82) := "Test variable for simulation - a command for the rotation of the basket is enabled";
  gc_DbmTranslation_fr_Text2160 : WSTRING(54) := "Test variable for simulation - turret angular position";
  gc_DbmTranslation_fr_Text2161 : WSTRING(82) := "Test variable for simulation - a command for the rotation of the turret is enabled";
  gc_DbmTranslation_fr_Text2162 : WSTRING(33) := "Turret is in the rear center zone";
  gc_DbmTranslation_fr_Text2163 : WSTRING(43) := "Turret is in the front positive center zone";
  gc_DbmTranslation_fr_Text2164 : WSTRING(43) := "Turret is in the front negative center zone";
  gc_DbmTranslation_fr_Text2165 : WSTRING(26) := "Basket in centrer position";
  gc_DbmTranslation_fr_Text2166 : WSTRING(31) := "Turret rotation command enabled";
  gc_DbmTranslation_fr_Text2167 : WSTRING(38) := "counter stop turret rotation for debug";
  gc_DbmTranslation_fr_Text2168 : WSTRING(41) := "counter no stop turret rotation for debug";
  gc_DbmTranslation_fr_Text2169 : WSTRING(63) := "Fonction active when commande neutre and button fucntion pushed";
  gc_DbmTranslation_fr_Text2170 : WSTRING(61) := "Command neutre when all command of TOR movement is not pushed";
  gc_DbmTranslation_fr_Text2171 : WSTRING(74) := "Authorize driving mast when fonction active and dead man pedal are actived";
  gc_DbmTranslation_fr_Text2172 : WSTRING(23) := "Folded position of mast";
  gc_DbmTranslation_fr_Text2173 : WSTRING(45) := "Stop all movement TOR when mast is sollicited";
  gc_DbmTranslation_fr_Text2174 : WSTRING(28) := "Raz distance traveled button";
  gc_DbmTranslation_fr_Text2175 : WSTRING(30) := "Distance traveled in milimeter";
  gc_DbmTranslation_fr_Text2176 : WSTRING(46) := "Delta beetween min and max encodeur mast value";
  gc_DbmTranslation_fr_Text2177 : WSTRING(48) := "Mast measure encodeur in cm additional to offset";
  gc_DbmTranslation_fr_Text2178 : WSTRING(27) := "Mast measure encodeur in cm";
  gc_DbmTranslation_fr_Text2179 : WSTRING(21) := "No movement is during";
  gc_DbmTranslation_fr_Text2180 : WSTRING(71) := "Scaling joystick mat , joytstick telescope is used to pilot mat measure";
  gc_DbmTranslation_fr_Text2181 : WSTRING(25) := "Time with mast not folded";
  gc_DbmTranslation_fr_Text2182 : WSTRING(56) := "Down axle oscillant when function mast measure is active";
  gc_DbmTranslation_fr_Text2183 : WSTRING(58) := "Flag to disply on scree distance traveled wth unfolded mat";
  gc_DbmTranslation_fr_Text2184 : WSTRING(22) := "Mast in upper position";
  gc_DbmTranslation_fr_Text2185 : WSTRING(23) := "Mast in folded position";
  gc_DbmTranslation_fr_Text2186 : WSTRING(27) := "Mast valve en down position";
  gc_DbmTranslation_fr_Text2187 : WSTRING(31) := "Post interdiction for mast SNCF";
  gc_DbmTranslation_fr_Text2188 : WSTRING(38) := "Memorisation of first valid cycle mast";
  gc_DbmTranslation_fr_Text2189 : WSTRING(33) := "Mast contact autorisation of mvts";
  gc_DbmTranslation_fr_Text2190 : WSTRING(39) := "Interdiction of Nacelle And Turret post";
  gc_DbmTranslation_fr_Text2191 : WSTRING(52) := "Warning picto for the first valid cycle of mast SNCF";
  gc_DbmTranslation_fr_Text2192 : WSTRING(53) := "offset mast in centimeter additional to scaling value";
  gc_DbmTranslation_fr_Text2193 : WSTRING(19) := "Folded mat treshold";
  gc_DbmTranslation_fr_Text2194 : WSTRING(30) := "Folded mat treshold hysterisys";
  gc_DbmTranslation_fr_Text2195 : WSTRING(51) := "Min calibration value of encodeut mast sensor value";
  gc_DbmTranslation_fr_Text2196 : WSTRING(51) := "Max calibration value of encodeut mast sensor value";
  gc_DbmTranslation_fr_Text2197 : WSTRING(52) := "Min calibration value of encodeut mast in centimeter";
  gc_DbmTranslation_fr_Text2198 : WSTRING(52) := "Max calibration value of encodeut mast in centimeter";
  gc_DbmTranslation_fr_Text2199 : WSTRING(91) := "Refresh cycle time or the mast digital display ( cycle time of the message sent to display)";
